(* Logix 5000 project; controller ACMI_PLC vendor 1 type 14 code 101 rev 19.11; software revision 19.01; part 2 of 18 *)

        [362].TIME.DAY := 6, [362].TIME.HOUR := 12, [362].TIME.MINUTE := 4, [362].TIME.SECOND := 14, [362].TIME.MICROSECOND := 99935, [362].EVENT := '2016/08/06   12:04:14   USER : PPS RESET FAULT BUTTON PRESSED', [363].TIME.YEAR := 2016, [363].TIME.MONTH := 8, [363].TIME.DAY := 6, [363].TIME.HOUR := 14, [363].TIME.MINUTE := 57, [363].TIME.SECOND := 32, [363].TIME.MICROSECOND := 599468, [363].EVENT := '2016/08/06   14:57:32   FAULT : QOW1 : Charge Outside Window Detected', [364].TIME.YEAR := 2016, [364].TIME.MONTH := 8, [364].TIME.DAY := 6, [364].TIME.HOUR := 14, [364].TIME.MINUTE := 57, [364].TIME.SECOND := 32, [364].TIME.MICROSECOND := 799580, [364].EVENT := '2016/08/06   14:57:32   USER : PPS RESET FAULT BUTTON PRESSED', [365].TIME.YEAR := 2016, [365].TIME.MONTH := 8, [365].TIME.DAY := 6, [365].TIME.HOUR := 14, [365].TIME.MINUTE := 57, [365].TIME.SECOND := 41, [365].TIME.MICROSECOND := 799582, [365].EVENT := '2016/08/06   14:57:41   USER : PPS RESET FAULT BUTTON PRESSED', [366].TIME.YEAR := 2016, [366].TIME.MONTH := 8, [366].TIME.DAY := 6, [366].TIME.HOUR := 14, [366].TIME.MINUTE := 57, [366].TIME.SECOND := 45, [366].TIME.MICROSECOND := 499509, [366].EVENT := '2016/08/06   14:57:45   USER : PPS RESET FAULT BUTTON PRESSED', [367].TIME.YEAR := 2016, [367].TIME.MONTH := 8, [367].TIME.DAY := 6, [367].TIME.HOUR := 18, [367].TIME.MINUTE := 23, [367].TIME.SECOND := 45, [367].TIME.MICROSECOND := 899510, [367].EVENT := '2016/08/06   18:23:45   USER : PPS RESET FAULT BUTTON PRESSED', [368].TIME.YEAR := 2016, [368].TIME.MONTH := 8, [368].TIME.DAY := 6, [368].TIME.HOUR := 18, [368].TIME.MINUTE := 28, [368].TIME.SECOND := 40, [368].TIME.MICROSECOND := 699977, [368].EVENT := '2016/08/06   18:28:40   FAULT : QOW1 : Charge Outside Window Detected', [369].TIME.YEAR := 2016, [369].TIME.MONTH := 8, [369].TIME.DAY := 6, [369].TIME.HOUR := 18, [369].TIME.MINUTE := 31, [369].TIME.SECOND := 49,
        [369].TIME.MICROSECOND := 299504, [369].EVENT := '2016/08/06   18:31:49   USER : PPS RESET FAULT BUTTON PRESSED', [370].TIME.YEAR := 2016, [370].TIME.MONTH := 8, [370].TIME.DAY := 7, [370].TIME.HOUR := 13, [370].TIME.MINUTE := 14, [370].TIME.SECOND := 49, [370].TIME.MICROSECOND := 699851, [370].EVENT := '2016/08/07   13:14:49   USER : PPS RESET FAULT BUTTON PRESSED', [371].TIME.YEAR := 2016, [371].TIME.MONTH := 8, [371].TIME.DAY := 7, [371].TIME.HOUR := 13, [371].TIME.MINUTE := 14, [371].TIME.SECOND := 53, [371].TIME.MICROSECOND := 399507, [371].EVENT := '2016/08/07   13:14:53   USER : PPS RESET FAULT BUTTON PRESSED', [372].TIME.YEAR := 2016, [372].TIME.MONTH := 8, [372].TIME.DAY := 7, [372].TIME.HOUR := 14, [372].TIME.MINUTE := 4, [372].TIME.SECOND := 34, [372].TIME.MICROSECOND := 499506, [372].EVENT := '2016/08/07   14:04:34   USER : PPS RESET FAULT BUTTON PRESSED', [373].TIME.YEAR := 2016, [373].TIME.MONTH := 8, [373].TIME.DAY := 7, [373].TIME.HOUR := 14, [373].TIME.MINUTE := 10, [373].TIME.SECOND := 33, [373].TIME.MICROSECOND := 599503, [373].EVENT := '2016/08/07   14:10:33   USER : PPS RESET FAULT BUTTON PRESSED', [374].TIME.YEAR := 2016, [374].TIME.MONTH := 8, [374].TIME.DAY := 7, [374].TIME.HOUR := 15, [374].TIME.MINUTE := 43, [374].TIME.SECOND := 5, [374].TIME.MICROSECOND := 599722, [374].EVENT := '2016/08/07   15:43:05   USER : PPS RESET FAULT BUTTON PRESSED', [375].TIME.YEAR := 2016, [375].TIME.MONTH := 8, [375].TIME.DAY := 7, [375].TIME.HOUR := 16, [375].TIME.MINUTE := 8, [375].TIME.SECOND := 27, [375].TIME.MICROSECOND := 699933, [375].EVENT := '2016/08/07   16:08:27   USER : PPS RESET FAULT BUTTON PRESSED', [376].TIME.YEAR := 2016, [376].TIME.MONTH := 8, [376].TIME.DAY := 7, [376].TIME.HOUR := 16, [376].TIME.MINUTE := 12, [376].TIME.SECOND := 25, [376].TIME.MICROSECOND := 299512, [376].EVENT := '2016/08/07   16:12:25   USER : PPS RESET FAULT BUTTON PRESSED', [377].TIME.YEAR := 2016, [377].TIME.MONTH := 8,
        [377].TIME.DAY := 7, [377].TIME.HOUR := 16, [377].TIME.MINUTE := 15, [377].TIME.SECOND := 37, [377].TIME.MICROSECOND := 299739, [377].EVENT := '2016/08/07   16:15:37   USER : PPS RESET FAULT BUTTON PRESSED', [378].TIME.YEAR := 2016, [378].TIME.MONTH := 8, [378].TIME.DAY := 7, [378].TIME.HOUR := 16, [378].TIME.MINUTE := 28, [378].TIME.SECOND := 37, [378].TIME.MICROSECOND := 299464, [378].EVENT := '2016/08/07   16:28:37   FAULT : QOW1 : Charge Outside Window Detected', [379].TIME.YEAR := 2016, [379].TIME.MONTH := 8, [379].TIME.DAY := 7, [379].TIME.HOUR := 16, [379].TIME.MINUTE := 29, [379].TIME.SECOND := 15, [379].TIME.MICROSECOND := 699509, [379].EVENT := '2016/08/07   16:29:15   USER : PPS RESET FAULT BUTTON PRESSED', [380].TIME.YEAR := 2016, [380].TIME.MONTH := 8, [380].TIME.DAY := 7, [380].TIME.HOUR := 16, [380].TIME.MINUTE := 29, [380].TIME.SECOND := 58, [380].TIME.MICROSECOND := 299502, [380].EVENT := '2016/08/07   16:29:58   USER : PPS RESET FAULT BUTTON PRESSED', [381].TIME.YEAR := 2016, [381].TIME.MONTH := 8, [381].TIME.DAY := 7, [381].TIME.HOUR := 17, [381].TIME.MINUTE := 7, [381].TIME.SECOND := 3, [381].TIME.MICROSECOND := 599449, [381].EVENT := '2016/08/07   17:07:03   FAULT : Storage Ring Accumulation HIGH', [382].TIME.YEAR := 2016, [382].TIME.MONTH := 8, [382].TIME.DAY := 7, [382].TIME.HOUR := 17, [382].TIME.MINUTE := 9, [382].TIME.SECOND := 13, [382].TIME.MICROSECOND := 499509, [382].EVENT := '2016/08/07   17:09:13   USER : PPS RESET FAULT BUTTON PRESSED', [383].TIME.YEAR := 2016, [383].TIME.MONTH := 8, [383].TIME.DAY := 7, [383].TIME.HOUR := 17, [383].TIME.MINUTE := 16, [383].TIME.SECOND := 23, [383].TIME.MICROSECOND := 799943, [383].EVENT := '2016/08/07   17:16:23   USER : PPS RESET FAULT BUTTON PRESSED', [384].TIME.YEAR := 2016, [384].TIME.MONTH := 8, [384].TIME.DAY := 7, [384].TIME.HOUR := 17, [384].TIME.MINUTE := 16, [384].TIME.SECOND := 25,
        [384].TIME.MICROSECOND := 699505, [384].EVENT := '2016/08/07   17:16:25   USER : PPS RESET FAULT BUTTON PRESSED', [385].TIME.YEAR := 2016, [385].TIME.MONTH := 8, [385].TIME.DAY := 7, [385].TIME.HOUR := 17, [385].TIME.MINUTE := 18, [385].TIME.SECOND := 4, [385].TIME.MICROSECOND := 899594, [385].EVENT := '2016/08/07   17:18:04   FAULT : Storage Ring Accumulation HIGH', [386].TIME.YEAR := 2016, [386].TIME.MONTH := 8, [386].TIME.DAY := 7, [386].TIME.HOUR := 17, [386].TIME.MINUTE := 18, [386].TIME.SECOND := 50, [386].TIME.MICROSECOND := 599506, [386].EVENT := '2016/08/07   17:18:50   USER : PPS RESET FAULT BUTTON PRESSED', [387].TIME.YEAR := 2016, [387].TIME.MONTH := 8, [387].TIME.DAY := 7, [387].TIME.HOUR := 17, [387].TIME.MINUTE := 20, [387].TIME.SECOND := 25, [387].TIME.MICROSECOND := 499450, [387].EVENT := '2016/08/07   17:20:25   FAULT : Storage Ring Accumulation HIGH', [388].TIME.YEAR := 2016, [388].TIME.MONTH := 8, [388].TIME.DAY := 7, [388].TIME.HOUR := 17, [388].TIME.MINUTE := 20, [388].TIME.SECOND := 25, [388].TIME.MICROSECOND := 699462, [388].EVENT := '2016/08/07   17:20:25   FAULT : QOW1 : Charge Outside Window Detected', [389].TIME.YEAR := 2016, [389].TIME.MONTH := 8, [389].TIME.DAY := 7, [389].TIME.HOUR := 17, [389].TIME.MINUTE := 21, [389].TIME.SECOND := 52, [389].TIME.MICROSECOND := 699506, [389].EVENT := '2016/08/07   17:21:52   USER : PPS RESET FAULT BUTTON PRESSED', [390].TIME.YEAR := 2016, [390].TIME.MONTH := 8, [390].TIME.DAY := 7, [390].TIME.HOUR := 17, [390].TIME.MINUTE := 30, [390].TIME.SECOND := 8, [390].TIME.MICROSECOND := 299449, [390].EVENT := '2016/08/07   17:30:08   FAULT : Storage Ring Accumulation HIGH', [391].TIME.YEAR := 2016, [391].TIME.MONTH := 8, [391].TIME.DAY := 7, [391].TIME.HOUR := 17, [391].TIME.MINUTE := 30, [391].TIME.SECOND := 53, [391].TIME.MICROSECOND := 299556, [391].EVENT := '2016/08/07   17:30:53   USER : PPS RESET FAULT BUTTON PRESSED', [392].TIME.YEAR := 2016, [392].TIME.MONTH := 8,
        [392].TIME.DAY := 7, [392].TIME.HOUR := 17, [392].TIME.MINUTE := 39, [392].TIME.SECOND := 26, [392].TIME.MICROSECOND := 699451, [392].EVENT := '2016/08/07   17:39:26   FAULT : Storage Ring Accumulation HIGH', [393].TIME.YEAR := 2016, [393].TIME.MONTH := 8, [393].TIME.DAY := 7, [393].TIME.HOUR := 17, [393].TIME.MINUTE := 40, [393].TIME.SECOND := 48, [393].TIME.MICROSECOND := 599508, [393].EVENT := '2016/08/07   17:40:48   USER : PPS RESET FAULT BUTTON PRESSED', [394].TIME.YEAR := 2016, [394].TIME.MONTH := 8, [394].TIME.DAY := 7, [394].TIME.HOUR := 17, [394].TIME.MINUTE := 40, [394].TIME.SECOND := 49, [394].TIME.MICROSECOND := 99507, [394].EVENT := '2016/08/07   17:40:49   USER : PPS RESET FAULT BUTTON PRESSED', [395].TIME.YEAR := 2016, [395].TIME.MONTH := 8, [395].TIME.DAY := 7, [395].TIME.HOUR := 17, [395].TIME.MINUTE := 52, [395].TIME.MICROSECOND := 599599, [395].EVENT := '2016/08/07   17:52:00   FAULT : Storage Ring Accumulation HIGH', [396].TIME.YEAR := 2016, [396].TIME.MONTH := 8, [396].TIME.DAY := 7, [396].TIME.HOUR := 17, [396].TIME.MINUTE := 53, [396].TIME.SECOND := 10, [396].TIME.MICROSECOND := 99562, [396].EVENT := '2016/08/07   17:53:10   USER : PPS RESET FAULT BUTTON PRESSED', [397].TIME.YEAR := 2016, [397].TIME.MONTH := 8, [397].TIME.DAY := 7, [397].TIME.HOUR := 18, [397].TIME.MICROSECOND := 999511, [397].EVENT := '2016/08/07   18:00:00   USER : PPS RESET FAULT BUTTON PRESSED', [398].TIME.YEAR := 2016, [398].TIME.MONTH := 8, [398].TIME.DAY := 7, [398].TIME.HOUR := 18, [398].TIME.SECOND := 51, [398].TIME.MICROSECOND := 499521, [398].EVENT := '2016/08/07   18:00:51   USER : PPS RESET FAULT BUTTON PRESSED', [399].TIME.YEAR := 2016, [399].TIME.MONTH := 8, [399].TIME.DAY := 7, [399].TIME.HOUR := 18, [399].TIME.MINUTE := 8, [399].TIME.SECOND := 30, [399].TIME.MICROSECOND := 299507, [399].EVENT := '2016/08/07   18:08:30   USER : PPS RESET FAULT BUTTON PRESSED', [400].TIME.YEAR := 2016, [400].TIME.MONTH := 8,
        [400].TIME.DAY := 8, [400].TIME.MINUTE := 42, [400].TIME.SECOND := 51, [400].TIME.MICROSECOND := 899938, [400].EVENT := '2016/08/08   00:42:51   USER : PPS RESET FAULT BUTTON PRESSED', [401].TIME.YEAR := 2016, [401].TIME.MONTH := 8, [401].TIME.DAY := 8, [401].TIME.HOUR := 1, [401].TIME.MINUTE := 23, [401].TIME.SECOND := 6, [401].TIME.MICROSECOND := 299510, [401].EVENT := '2016/08/08   01:23:06   USER : PPS RESET FAULT BUTTON PRESSED', [402].TIME.YEAR := 2016, [402].TIME.MONTH := 8, [402].TIME.DAY := 8, [402].TIME.HOUR := 4, [402].TIME.MINUTE := 37, [402].TIME.SECOND := 22, [402].TIME.MICROSECOND := 699521, [402].EVENT := '2016/08/08   04:37:22   USER : PPS RESET FAULT BUTTON PRESSED', [403].TIME.YEAR := 2016, [403].TIME.MONTH := 8, [403].TIME.DAY := 8, [403].TIME.HOUR := 8, [403].TIME.MINUTE := 26, [403].TIME.SECOND := 45, [403].TIME.MICROSECOND := 170, [403].EVENT := '2016/08/08   08:26:45   USER : PPS RESET FAULT BUTTON PRESSED', [404].TIME.YEAR := 2016, [404].TIME.MONTH := 8, [404].TIME.DAY := 8, [404].TIME.HOUR := 14, [404].TIME.MINUTE := 8, [404].TIME.SECOND := 27, [404].TIME.MICROSECOND := 399526, [404].EVENT := '2016/08/08   14:08:27   USER : PPS RESET FAULT BUTTON PRESSED', [405].TIME.YEAR := 2016, [405].TIME.MONTH := 8, [405].TIME.DAY := 8, [405].TIME.HOUR := 16, [405].TIME.MINUTE := 58, [405].TIME.SECOND := 17, [405].TIME.MICROSECOND := 299507, [405].EVENT := '2016/08/08   16:58:17   USER : PPS RESET FAULT BUTTON PRESSED', [406].TIME.YEAR := 2016, [406].TIME.MONTH := 8, [406].TIME.DAY := 8, [406].TIME.HOUR := 20, [406].TIME.MINUTE := 53, [406].TIME.SECOND := 34, [406].TIME.MICROSECOND := 99465, [406].EVENT := '2016/08/08   20:53:34   FAULT : QOW1 : Charge Outside Window Detected', [407].TIME.YEAR := 2016, [407].TIME.MONTH := 8, [407].TIME.DAY := 8, [407].TIME.HOUR := 20, [407].TIME.MINUTE := 53, [407].TIME.SECOND := 50, [407].TIME.MICROSECOND := 299514,
        [407].EVENT := '2016/08/08   20:53:50   USER : PPS RESET FAULT BUTTON PRESSED', [408].TIME.YEAR := 2016, [408].TIME.MONTH := 8, [408].TIME.DAY := 8, [408].TIME.HOUR := 21, [408].TIME.SECOND := 58, [408].TIME.MICROSECOND := 799510, [408].EVENT := '2016/08/08   21:00:58   USER : PPS RESET FAULT BUTTON PRESSED', [409].TIME.YEAR := 2016, [409].TIME.MONTH := 8, [409].TIME.DAY := 9, [409].TIME.HOUR := 16, [409].TIME.MINUTE := 51, [409].TIME.SECOND := 48, [409].TIME.MICROSECOND := 699509, [409].EVENT := '2016/08/09   16:51:48   USER : PPS RESET FAULT BUTTON PRESSED', [410].TIME.YEAR := 2016, [410].TIME.MONTH := 8, [410].TIME.DAY := 9, [410].TIME.HOUR := 16, [410].TIME.MINUTE := 52, [410].TIME.SECOND := 16, [410].TIME.MICROSECOND := 999461, [410].EVENT := '2016/08/09   16:52:16   FAULT : QOW1 : Charge Outside Window Detected', [411].TIME.YEAR := 2016, [411].TIME.MONTH := 8, [411].TIME.DAY := 9, [411].TIME.HOUR := 16, [411].TIME.MINUTE := 52, [411].TIME.SECOND := 51, [411].TIME.MICROSECOND := 199503, [411].EVENT := '2016/08/09   16:52:51   USER : PPS RESET FAULT BUTTON PRESSED', [412].TIME.YEAR := 2016, [412].TIME.MONTH := 8, [412].TIME.DAY := 9, [412].TIME.HOUR := 18, [412].TIME.MINUTE := 25, [412].TIME.SECOND := 25, [412].TIME.MICROSECOND := 799513, [412].EVENT := '2016/08/09   18:25:25   USER : PPS RESET FAULT BUTTON PRESSED', [413].TIME.YEAR := 2016, [413].TIME.MONTH := 8, [413].TIME.DAY := 9, [413].TIME.HOUR := 18, [413].TIME.MINUTE := 44, [413].TIME.SECOND := 50, [413].TIME.MICROSECOND := 600033, [413].EVENT := '2016/08/09   18:44:50   USER : PPS RESET FAULT BUTTON PRESSED', [414].TIME.YEAR := 2016, [414].TIME.MONTH := 8, [414].TIME.DAY := 9, [414].TIME.HOUR := 22, [414].TIME.MINUTE := 53, [414].TIME.SECOND := 46, [414].TIME.MICROSECOND := 999841, [414].EVENT := '2016/08/09   22:53:46   FAULT : QOW1 : Charge Outside Window Detected', [415].TIME.YEAR := 2016, [415].TIME.MONTH := 8, [415].TIME.DAY := 9, [415].TIME.HOUR := 22,
        [415].TIME.MINUTE := 54, [415].TIME.SECOND := 3, [415].TIME.MICROSECOND := 99504, [415].EVENT := '2016/08/09   22:54:03   USER : PPS RESET FAULT BUTTON PRESSED', [416].TIME.YEAR := 2016, [416].TIME.MONTH := 8, [416].TIME.DAY := 10, [416].TIME.HOUR := 4, [416].TIME.MINUTE := 15, [416].TIME.SECOND := 3, [416].TIME.MICROSECOND := 899896, [416].EVENT := '2016/08/10   04:15:03   FAULT : QOW1 : Charge Outside Window Detected', [417].TIME.YEAR := 2016, [417].TIME.MONTH := 8, [417].TIME.DAY := 10, [417].TIME.HOUR := 4, [417].TIME.MINUTE := 15, [417].TIME.SECOND := 18, [417].TIME.MICROSECOND := 799507, [417].EVENT := '2016/08/10   04:15:18   USER : PPS RESET FAULT BUTTON PRESSED', [418].TIME.YEAR := 2016, [418].TIME.MONTH := 8, [418].TIME.DAY := 10, [418].TIME.HOUR := 17, [418].TIME.MINUTE := 5, [418].TIME.SECOND := 50, [418].TIME.MICROSECOND := 799512, [418].EVENT := '2016/08/10   17:05:50   FAULT : QOW1 : Charge Outside Window Detected', [419].TIME.YEAR := 2016, [419].TIME.MONTH := 8, [419].TIME.DAY := 10, [419].TIME.HOUR := 17, [419].TIME.MINUTE := 5, [419].TIME.SECOND := 51, [419].TIME.MICROSECOND := 99507, [419].EVENT := '2016/08/10   17:05:51   USER : PPS RESET FAULT BUTTON PRESSED', [420].TIME.YEAR := 2016, [420].TIME.MONTH := 8, [420].TIME.DAY := 10, [420].TIME.HOUR := 17, [420].TIME.MINUTE := 6, [420].TIME.SECOND := 1, [420].TIME.MICROSECOND := 100028, [420].EVENT := '2016/08/10   17:06:01   USER : PPS RESET FAULT BUTTON PRESSED', [421].TIME.YEAR := 2016, [421].TIME.MONTH := 8, [421].TIME.DAY := 10, [421].TIME.HOUR := 17, [421].TIME.MINUTE := 8, [421].TIME.SECOND := 33, [421].TIME.MICROSECOND := 599516, [421].EVENT := '2016/08/10   17:08:33   USER : PPS RESET FAULT BUTTON PRESSED', [422].TIME.YEAR := 2016, [422].TIME.MONTH := 8, [422].TIME.DAY := 10, [422].TIME.HOUR := 17, [422].TIME.MINUTE := 33, [422].TIME.SECOND := 25, [422].TIME.MICROSECOND := 299511, [422].EVENT := '2016/08/10   17:33:25   USER : PPS RESET FAULT BUTTON PRESSED',
        [423].TIME.YEAR := 2016, [423].TIME.MONTH := 8, [423].TIME.DAY := 10, [423].TIME.HOUR := 17, [423].TIME.MINUTE := 46, [423].TIME.SECOND := 7, [423].TIME.MICROSECOND := 799463, [423].EVENT := '2016/08/10   17:46:07   FAULT : QOW1 : Charge Outside Window Detected', [424].TIME.YEAR := 2016, [424].TIME.MONTH := 8, [424].TIME.DAY := 10, [424].TIME.HOUR := 17, [424].TIME.MINUTE := 47, [424].TIME.SECOND := 1, [424].TIME.MICROSECOND := 599530, [424].EVENT := '2016/08/10   17:47:01   USER : PPS RESET FAULT BUTTON PRESSED', [425].TIME.YEAR := 2016, [425].TIME.MONTH := 8, [425].TIME.DAY := 11, [425].TIME.HOUR := 1, [425].TIME.MINUTE := 16, [425].TIME.SECOND := 30, [425].TIME.MICROSECOND := 999451, [425].EVENT := '2016/08/11   01:16:30   FAULT : Storage Ring Accumulation HIGH', [426].TIME.YEAR := 2016, [426].TIME.MONTH := 8, [426].TIME.DAY := 11, [426].TIME.HOUR := 1, [426].TIME.MINUTE := 16, [426].TIME.SECOND := 55, [426].TIME.MICROSECOND := 99506, [426].EVENT := '2016/08/11   01:16:55   USER : PPS RESET FAULT BUTTON PRESSED', [427].TIME.YEAR := 2016, [427].TIME.MONTH := 8, [427].TIME.DAY := 11, [427].TIME.HOUR := 5, [427].TIME.MINUTE := 52, [427].TIME.SECOND := 19, [427].TIME.MICROSECOND := 499510, [427].EVENT := '2016/08/11   05:52:19   USER : PPS RESET FAULT BUTTON PRESSED', [428].TIME.YEAR := 2016, [428].TIME.MONTH := 8, [428].TIME.DAY := 11, [428].TIME.HOUR := 6, [428].TIME.MINUTE := 51, [428].TIME.SECOND := 51, [428].TIME.MICROSECOND := 499508, [428].EVENT := '2016/08/11   06:51:51   USER : PPS RESET FAULT BUTTON PRESSED', [429].TIME.YEAR := 2016, [429].TIME.MONTH := 8, [429].TIME.DAY := 11, [429].TIME.HOUR := 13, [429].TIME.MINUTE := 21, [429].TIME.SECOND := 20, [429].TIME.MICROSECOND := 699504, [429].EVENT := '2016/08/11   13:21:20   USER : PPS RESET FAULT BUTTON PRESSED', [430].TIME.YEAR := 2016, [430].TIME.MONTH := 8, [430].TIME.DAY := 11, [430].TIME.HOUR := 14,
        [430].TIME.MINUTE := 4, [430].TIME.SECOND := 47, [430].TIME.MICROSECOND := 599502, [430].EVENT := '2016/08/11   14:04:47   USER : PPS RESET FAULT BUTTON PRESSED', [431].TIME.YEAR := 2016, [431].TIME.MONTH := 8, [431].TIME.DAY := 11, [431].TIME.HOUR := 15, [431].TIME.MINUTE := 12, [431].TIME.SECOND := 47, [431].TIME.MICROSECOND := 999508, [431].EVENT := '2016/08/11   15:12:47   USER : PPS RESET FAULT BUTTON PRESSED', [432].TIME.YEAR := 2016, [432].TIME.MONTH := 8, [432].TIME.DAY := 11, [432].TIME.HOUR := 19, [432].TIME.MINUTE := 47, [432].TIME.SECOND := 25, [432].TIME.MICROSECOND := 999651, [432].EVENT := '2016/08/11   19:47:25   USER : PPS RESET FAULT BUTTON PRESSED', [433].TIME.YEAR := 2016, [433].TIME.MONTH := 8, [433].TIME.DAY := 12, [433].TIME.HOUR := 2, [433].TIME.MINUTE := 31, [433].TIME.SECOND := 8, [433].TIME.MICROSECOND := 399504, [433].EVENT := '2016/08/12   02:31:08   USER : PPS RESET FAULT BUTTON PRESSED', [434].TIME.YEAR := 2016, [434].TIME.MONTH := 8, [434].TIME.DAY := 12, [434].TIME.HOUR := 16, [434].TIME.MINUTE := 21, [434].TIME.SECOND := 30, [434].TIME.MICROSECOND := 499936, [434].EVENT := '2016/08/12   16:21:30   USER : PPS RESET FAULT BUTTON PRESSED', [435].TIME.YEAR := 2016, [435].TIME.MONTH := 8, [435].TIME.DAY := 12, [435].TIME.HOUR := 16, [435].TIME.MINUTE := 21, [435].TIME.SECOND := 54, [435].TIME.MICROSECOND := 899511, [435].EVENT := '2016/08/12   16:21:54   USER : PPS RESET FAULT BUTTON PRESSED', [436].TIME.YEAR := 2016, [436].TIME.MONTH := 8, [436].TIME.DAY := 12, [436].TIME.HOUR := 16, [436].TIME.MINUTE := 24, [436].TIME.MICROSECOND := 99513, [436].EVENT := '2016/08/12   16:24:00   USER : PPS RESET FAULT BUTTON PRESSED', [437].TIME.YEAR := 2016, [437].TIME.MONTH := 8, [437].TIME.DAY := 12, [437].TIME.HOUR := 16, [437].TIME.MINUTE := 32, [437].TIME.SECOND := 10, [437].TIME.MICROSECOND := 99511, [437].EVENT := '2016/08/12   16:32:10   USER : PPS RESET FAULT BUTTON PRESSED', [438].TIME.YEAR := 2016,
        [438].TIME.MONTH := 8, [438].TIME.DAY := 12, [438].TIME.HOUR := 16, [438].TIME.MINUTE := 52, [438].TIME.SECOND := 35, [438].TIME.MICROSECOND := 999515, [438].EVENT := '2016/08/12   16:52:35   FAULT : QOW1 : Charge Outside Window Detected', [439].TIME.YEAR := 2016, [439].TIME.MONTH := 8, [439].TIME.DAY := 12, [439].TIME.HOUR := 16, [439].TIME.MINUTE := 57, [439].TIME.SECOND := 19, [439].TIME.MICROSECOND := 99507, [439].EVENT := '2016/08/12   16:57:19   USER : PPS RESET FAULT BUTTON PRESSED', [440].TIME.YEAR := 2016, [440].TIME.MONTH := 8, [440].TIME.DAY := 13, [440].TIME.HOUR := 10, [440].TIME.MINUTE := 42, [440].TIME.SECOND := 33, [440].TIME.MICROSECOND := 199466, [440].EVENT := '2016/08/13   10:42:33   FAULT : QOW1 : Charge Outside Window Detected', [441].TIME.YEAR := 2016, [441].TIME.MONTH := 8, [441].TIME.DAY := 13, [441].TIME.HOUR := 10, [441].TIME.MINUTE := 43, [441].TIME.SECOND := 44, [441].TIME.MICROSECOND := 299504, [441].EVENT := '2016/08/13   10:43:44   USER : PPS RESET FAULT BUTTON PRESSED', [442].TIME.YEAR := 2016, [442].TIME.MONTH := 8, [442].TIME.DAY := 13, [442].TIME.HOUR := 10, [442].TIME.MINUTE := 43, [442].TIME.SECOND := 46, [442].TIME.MICROSECOND := 499651, [442].EVENT := '2016/08/13   10:43:46   USER : PPS RESET FAULT BUTTON PRESSED', [443].TIME.YEAR := 2016, [443].TIME.MONTH := 8, [443].TIME.DAY := 13, [443].TIME.HOUR := 18, [443].TIME.MINUTE := 25, [443].TIME.SECOND := 45, [443].TIME.MICROSECOND := 200030, [443].EVENT := '2016/08/13   18:25:45   USER : PPS RESET FAULT BUTTON PRESSED', [444].TIME.YEAR := 2016, [444].TIME.MONTH := 8, [444].TIME.DAY := 13, [444].TIME.HOUR := 19, [444].TIME.MINUTE := 6, [444].TIME.SECOND := 5, [444].TIME.MICROSECOND := 499509, [444].EVENT := '2016/08/13   19:06:05   USER : PPS RESET FAULT BUTTON PRESSED', [445].TIME.YEAR := 2016, [445].TIME.MONTH := 8, [445].TIME.DAY := 13, [445].TIME.HOUR := 19, [445].TIME.MINUTE := 7,
        [445].TIME.SECOND := 19, [445].TIME.MICROSECOND := 899509, [445].EVENT := '2016/08/13   19:07:19   USER : PPS RESET FAULT BUTTON PRESSED', [446].TIME.YEAR := 2016, [446].TIME.MONTH := 8, [446].TIME.DAY := 13, [446].TIME.HOUR := 21, [446].TIME.MINUTE := 17, [446].TIME.SECOND := 33, [446].TIME.MICROSECOND := 699513, [446].EVENT := '2016/08/13   21:17:33   USER : PPS RESET FAULT BUTTON PRESSED', [447].TIME.YEAR := 2016, [447].TIME.MONTH := 8, [447].TIME.DAY := 14, [447].TIME.HOUR := 3, [447].TIME.MINUTE := 19, [447].TIME.SECOND := 29, [447].TIME.MICROSECOND := 199465, [447].EVENT := '2016/08/14   03:19:29   FAULT : QOW1 : Charge Outside Window Detected', [448].TIME.YEAR := 2016, [448].TIME.MONTH := 8, [448].TIME.DAY := 14, [448].TIME.HOUR := 3, [448].TIME.MINUTE := 30, [448].TIME.SECOND := 16, [448].TIME.MICROSECOND := 699503, [448].EVENT := '2016/08/14   03:30:16   USER : PPS RESET FAULT BUTTON PRESSED', [449].TIME.YEAR := 2016, [449].TIME.MONTH := 8, [449].TIME.DAY := 14, [449].TIME.HOUR := 3, [449].TIME.MINUTE := 38, [449].TIME.SECOND := 57, [449].TIME.MICROSECOND := 999680, [449].EVENT := '2016/08/14   03:38:57   USER : PPS RESET FAULT BUTTON PRESSED', [450].TIME.YEAR := 2016, [450].TIME.MONTH := 8, [450].TIME.DAY := 14, [450].TIME.HOUR := 3, [450].TIME.MINUTE := 39, [450].TIME.SECOND := 19, [450].TIME.MICROSECOND := 999887, [450].EVENT := '2016/08/14   03:39:19   FAULT : QOW1 : Charge Outside Window Detected', [451].TIME.YEAR := 2016, [451].TIME.MONTH := 8, [451].TIME.DAY := 14, [451].TIME.HOUR := 3, [451].TIME.MINUTE := 58, [451].TIME.SECOND := 14, [451].TIME.MICROSECOND := 499507, [451].EVENT := '2016/08/14   03:58:14   USER : PPS RESET FAULT BUTTON PRESSED', [452].TIME.YEAR := 2016, [452].TIME.MONTH := 8, [452].TIME.DAY := 14, [452].TIME.HOUR := 4, [452].TIME.MINUTE := 1, [452].TIME.SECOND := 42, [452].TIME.MICROSECOND := 999504, [452].EVENT := '2016/08/14   04:01:42   USER : PPS RESET FAULT BUTTON PRESSED', [453].TIME.YEAR := 2016,
        [453].TIME.MONTH := 8, [453].TIME.DAY := 14, [453].TIME.HOUR := 9, [453].TIME.MINUTE := 12, [453].TIME.SECOND := 1, [453].TIME.MICROSECOND := 399505, [453].EVENT := '2016/08/14   09:12:01   USER : PPS RESET FAULT BUTTON PRESSED', [454].TIME.YEAR := 2016, [454].TIME.MONTH := 8, [454].TIME.DAY := 14, [454].TIME.HOUR := 9, [454].TIME.MINUTE := 12, [454].TIME.SECOND := 5, [454].TIME.MICROSECOND := 799506, [454].EVENT := '2016/08/14   09:12:05   USER : PPS RESET FAULT BUTTON PRESSED', [455].TIME.YEAR := 2016, [455].TIME.MONTH := 8, [455].TIME.DAY := 14, [455].TIME.HOUR := 19, [455].TIME.MINUTE := 56, [455].TIME.SECOND := 57, [455].TIME.MICROSECOND := 899462, [455].EVENT := '2016/08/14   19:56:57   FAULT : QOW1 : Charge Outside Window Detected', [456].TIME.YEAR := 2016, [456].TIME.MONTH := 8, [456].TIME.DAY := 14, [456].TIME.HOUR := 19, [456].TIME.MINUTE := 58, [456].TIME.SECOND := 49, [456].TIME.MICROSECOND := 999510, [456].EVENT := '2016/08/14   19:58:49   USER : PPS RESET FAULT BUTTON PRESSED', [457].TIME.YEAR := 2016, [457].TIME.MONTH := 8, [457].TIME.DAY := 14, [457].TIME.HOUR := 19, [457].TIME.MINUTE := 58, [457].TIME.SECOND := 55, [457].TIME.MICROSECOND := 999511, [457].EVENT := '2016/08/14   19:58:55   USER : PPS RESET FAULT BUTTON PRESSED', [458].TIME.YEAR := 2016, [458].TIME.MONTH := 8, [458].TIME.DAY := 15, [458].TIME.HOUR := 4, [458].TIME.MINUTE := 21, [458].TIME.SECOND := 30, [458].TIME.MICROSECOND := 299561, [458].EVENT := '2016/08/15   04:21:30   USER : PPS RESET FAULT BUTTON PRESSED', [459].TIME.YEAR := 2016, [459].TIME.MONTH := 8, [459].TIME.DAY := 16, [459].TIME.HOUR := 14, [459].TIME.MINUTE := 25, [459].TIME.SECOND := 39, [459].TIME.MICROSECOND := 699467, [459].EVENT := '2016/08/16   14:25:39   FAULT : QOW1 : Charge Outside Window Detected', [460].TIME.YEAR := 2016, [460].TIME.MONTH := 8, [460].TIME.DAY := 16, [460].TIME.HOUR := 14, [460].TIME.MINUTE := 25,
        [460].TIME.SECOND := 51, [460].TIME.MICROSECOND := 899506, [460].EVENT := '2016/08/16   14:25:51   USER : PPS RESET FAULT BUTTON PRESSED', [461].TIME.YEAR := 2016, [461].TIME.MONTH := 8, [461].TIME.DAY := 17, [461].TIME.HOUR := 9, [461].TIME.MINUTE := 19, [461].TIME.SECOND := 27, [461].TIME.MICROSECOND := 800026, [461].EVENT := '2016/08/17   09:19:27   USER : PPS RESET FAULT BUTTON PRESSED', [462].TIME.YEAR := 2016, [462].TIME.MONTH := 8, [462].TIME.DAY := 17, [462].TIME.HOUR := 9, [462].TIME.MINUTE := 29, [462].TIME.SECOND := 22, [462].TIME.MICROSECOND := 699555, [462].EVENT := '2016/08/17   09:29:22   USER : PPS RESET FAULT BUTTON PRESSED', [463].TIME.YEAR := 2016, [463].TIME.MONTH := 8, [463].TIME.DAY := 17, [463].TIME.HOUR := 9, [463].TIME.MINUTE := 30, [463].TIME.SECOND := 56, [463].TIME.MICROSECOND := 499725, [463].EVENT := '2016/08/17   09:30:56   USER : PPS RESET FAULT BUTTON PRESSED', [464].TIME.YEAR := 2016, [464].TIME.MONTH := 8, [464].TIME.DAY := 17, [464].TIME.HOUR := 9, [464].TIME.MINUTE := 45, [464].TIME.SECOND := 1, [464].TIME.MICROSECOND := 599506, [464].EVENT := '2016/08/17   09:45:01   USER : PPS RESET FAULT BUTTON PRESSED', [465].TIME.YEAR := 2016, [465].TIME.MONTH := 8, [465].TIME.DAY := 17, [465].TIME.HOUR := 10, [465].TIME.MINUTE := 8, [465].TIME.SECOND := 31, [465].TIME.MICROSECOND := 299511, [465].EVENT := '2016/08/17   10:08:31   USER : PPS RESET FAULT BUTTON PRESSED', [466].TIME.YEAR := 2016, [466].TIME.MONTH := 8, [466].TIME.DAY := 17, [466].TIME.HOUR := 10, [466].TIME.MINUTE := 12, [466].TIME.SECOND := 27, [466].TIME.MICROSECOND := 299510, [466].EVENT := '2016/08/17   10:12:27   USER : PPS RESET FAULT BUTTON PRESSED', [467].TIME.YEAR := 2016, [467].TIME.MONTH := 8, [467].TIME.DAY := 17, [467].TIME.HOUR := 10, [467].TIME.MINUTE := 12, [467].TIME.SECOND := 30, [467].TIME.MICROSECOND := 399508, [467].EVENT := '2016/08/17   10:12:30   USER : PPS RESET FAULT BUTTON PRESSED', [468].TIME.YEAR := 2016,
        [468].TIME.MONTH := 8, [468].TIME.DAY := 17, [468].TIME.HOUR := 10, [468].TIME.MINUTE := 12, [468].TIME.SECOND := 36, [468].TIME.MICROSECOND := 900030, [468].EVENT := '2016/08/17   10:12:36   USER : PPS RESET FAULT BUTTON PRESSED', [469].TIME.YEAR := 2016, [469].TIME.MONTH := 8, [469].TIME.DAY := 17, [469].TIME.HOUR := 10, [469].TIME.MINUTE := 17, [469].TIME.SECOND := 56, [469].TIME.MICROSECOND := 599509, [469].EVENT := '2016/08/17   10:17:56   USER : PPS RESET FAULT BUTTON PRESSED', [470].TIME.YEAR := 2016, [470].TIME.MONTH := 8, [470].TIME.DAY := 17, [470].TIME.HOUR := 11, [470].TIME.MINUTE := 20, [470].TIME.SECOND := 16, [470].TIME.MICROSECOND := 599503, [470].EVENT := '2016/08/17   11:20:16   USER : PPS RESET FAULT BUTTON PRESSED', [471].TIME.YEAR := 2016, [471].TIME.MONTH := 8, [471].TIME.DAY := 17, [471].TIME.HOUR := 11, [471].TIME.MINUTE := 20, [471].TIME.SECOND := 24, [471].TIME.MICROSECOND := 199526, [471].EVENT := '2016/08/17   11:20:24   USER : PPS RESET FAULT BUTTON PRESSED', [472].TIME.YEAR := 2016, [472].TIME.MONTH := 8, [472].TIME.DAY := 17, [472].TIME.HOUR := 11, [472].TIME.MINUTE := 22, [472].TIME.SECOND := 56, [472].TIME.MICROSECOND := 499504, [472].EVENT := '2016/08/17   11:22:56   USER : PPS RESET FAULT BUTTON PRESSED', [473].TIME.YEAR := 2016, [473].TIME.MONTH := 8, [473].TIME.DAY := 17, [473].TIME.HOUR := 11, [473].TIME.MINUTE := 24, [473].TIME.SECOND := 41, [473].TIME.MICROSECOND := 499557, [473].EVENT := '2016/08/17   11:24:41   USER : PPS RESET FAULT BUTTON PRESSED', [474].TIME.YEAR := 2016, [474].TIME.MONTH := 8, [474].TIME.DAY := 17, [474].TIME.HOUR := 13, [474].TIME.MINUTE := 2, [474].TIME.SECOND := 51, [474].TIME.MICROSECOND := 199488, [474].EVENT := '2016/08/17   13:02:51   FAULT : QOW1 : Charge Outside Window Detected', [475].TIME.YEAR := 2016, [475].TIME.MONTH := 8, [475].TIME.DAY := 17, [475].TIME.HOUR := 13, [475].TIME.MINUTE := 9,
        [475].TIME.SECOND := 21, [475].TIME.MICROSECOND := 500025, [475].EVENT := '2016/08/17   13:09:21   USER : PPS RESET FAULT BUTTON PRESSED', [476].TIME.YEAR := 2016, [476].TIME.MONTH := 8, [476].TIME.DAY := 17, [476].TIME.HOUR := 16, [476].TIME.MINUTE := 31, [476].TIME.SECOND := 24, [476].TIME.MICROSECOND := 999509, [476].EVENT := '2016/08/17   16:31:24   USER : PPS RESET FAULT BUTTON PRESSED', [477].TIME.YEAR := 2016, [477].TIME.MONTH := 8, [477].TIME.DAY := 17, [477].TIME.HOUR := 16, [477].TIME.MINUTE := 40, [477].TIME.SECOND := 51, [477].TIME.MICROSECOND := 299937, [477].EVENT := '2016/08/17   16:40:51   USER : PPS RESET FAULT BUTTON PRESSED', [478].TIME.YEAR := 2016, [478].TIME.MONTH := 8, [478].TIME.DAY := 17, [478].TIME.HOUR := 16, [478].TIME.MINUTE := 45, [478].TIME.SECOND := 7, [478].TIME.MICROSECOND := 199517, [478].EVENT := '2016/08/17   16:45:07   USER : PPS RESET FAULT BUTTON PRESSED', [479].TIME.YEAR := 2016, [479].TIME.MONTH := 8, [479].TIME.DAY := 17, [479].TIME.HOUR := 16, [479].TIME.MINUTE := 58, [479].TIME.SECOND := 20, [479].TIME.MICROSECOND := 899461, [479].EVENT := '2016/08/17   16:58:20   FAULT : QOW1 : Charge Outside Window Detected', [480].TIME.YEAR := 2016, [480].TIME.MONTH := 8, [480].TIME.DAY := 17, [480].TIME.HOUR := 17, [480].TIME.MINUTE := 2, [480].TIME.SECOND := 11, [480].TIME.MICROSECOND := 499503, [480].EVENT := '2016/08/17   17:02:11   USER : PPS RESET FAULT BUTTON PRESSED', [481].TIME.YEAR := 2016, [481].TIME.MONTH := 8, [481].TIME.DAY := 17, [481].TIME.HOUR := 17, [481].TIME.MINUTE := 2, [481].TIME.SECOND := 12, [481].TIME.MICROSECOND := 399510, [481].EVENT := '2016/08/17   17:02:12   USER : PPS RESET FAULT BUTTON PRESSED', [482].TIME.YEAR := 2016, [482].TIME.MONTH := 8, [482].TIME.DAY := 17, [482].TIME.HOUR := 17, [482].TIME.MINUTE := 32, [482].TIME.SECOND := 54, [482].TIME.MICROSECOND := 299505, [482].EVENT := '2016/08/17   17:32:54   USER : PPS RESET FAULT BUTTON PRESSED', [483].TIME.YEAR := 2016,
        [483].TIME.MONTH := 8, [483].TIME.DAY := 17, [483].TIME.HOUR := 17, [483].TIME.MINUTE := 34, [483].TIME.SECOND := 9, [483].TIME.MICROSECOND := 699506, [483].EVENT := '2016/08/17   17:34:09   USER : PPS RESET FAULT BUTTON PRESSED', [484].TIME.YEAR := 2016, [484].TIME.MONTH := 8, [484].TIME.DAY := 17, [484].TIME.HOUR := 18, [484].TIME.MINUTE := 32, [484].TIME.SECOND := 24, [484].TIME.MICROSECOND := 99507, [484].EVENT := '2016/08/17   18:32:24   USER : PPS RESET FAULT BUTTON PRESSED', [485].TIME.YEAR := 2016, [485].TIME.MONTH := 8, [485].TIME.DAY := 17, [485].TIME.HOUR := 20, [485].TIME.MINUTE := 51, [485].TIME.SECOND := 28, [485].TIME.MICROSECOND := 899507, [485].EVENT := '2016/08/17   20:51:28   USER : PPS RESET FAULT BUTTON PRESSED', [486].TIME.YEAR := 2016, [486].TIME.MONTH := 8, [486].TIME.DAY := 18, [486].TIME.MINUTE := 22, [486].TIME.SECOND := 47, [486].TIME.MICROSECOND := 799507, [486].EVENT := '2016/08/18   00:22:47   USER : PPS RESET FAULT BUTTON PRESSED', [487].TIME.YEAR := 2016, [487].TIME.MONTH := 8, [487].TIME.DAY := 18, [487].TIME.HOUR := 5, [487].TIME.MINUTE := 45, [487].TIME.SECOND := 44, [487].TIME.MICROSECOND := 399510, [487].EVENT := '2016/08/18   05:45:44   USER : PPS RESET FAULT BUTTON PRESSED', [488].TIME.YEAR := 2016, [488].TIME.MONTH := 8, [488].TIME.DAY := 18, [488].TIME.HOUR := 5, [488].TIME.MINUTE := 53, [488].TIME.SECOND := 55, [488].TIME.MICROSECOND := 599934, [488].EVENT := '2016/08/18   05:53:55   USER : PPS RESET FAULT BUTTON PRESSED', [489].TIME.YEAR := 2016, [489].TIME.MONTH := 8, [489].TIME.DAY := 18, [489].TIME.HOUR := 6, [489].TIME.MINUTE := 14, [489].TIME.SECOND := 56, [489].TIME.MICROSECOND := 599506, [489].EVENT := '2016/08/18   06:14:56   USER : PPS RESET FAULT BUTTON PRESSED', [490].TIME.YEAR := 2016, [490].TIME.MONTH := 8, [490].TIME.DAY := 18, [490].TIME.HOUR := 6, [490].TIME.MINUTE := 14, [490].TIME.SECOND := 58,
        [490].TIME.MICROSECOND := 99512, [490].EVENT := '2016/08/18   06:14:58   USER : PPS RESET FAULT BUTTON PRESSED', [491].TIME.YEAR := 2016, [491].TIME.MONTH := 8, [491].TIME.DAY := 18, [491].TIME.HOUR := 6, [491].TIME.MINUTE := 15, [491].TIME.SECOND := 1, [491].TIME.MICROSECOND := 999506, [491].EVENT := '2016/08/18   06:15:01   USER : PPS RESET FAULT BUTTON PRESSED', [492].TIME.YEAR := 2016, [492].TIME.MONTH := 8, [492].TIME.DAY := 18, [492].TIME.HOUR := 6, [492].TIME.MINUTE := 39, [492].TIME.SECOND := 58, [492].TIME.MICROSECOND := 799939, [492].EVENT := '2016/08/18   06:39:58   USER : PPS RESET FAULT BUTTON PRESSED', [493].TIME.YEAR := 2016, [493].TIME.MONTH := 8, [493].TIME.DAY := 19, [493].TIME.HOUR := 2, [493].TIME.MINUTE := 29, [493].TIME.SECOND := 21, [493].TIME.MICROSECOND := 599508, [493].EVENT := '2016/08/19   02:29:21   USER : PPS RESET FAULT BUTTON PRESSED', [494].TIME.YEAR := 2016, [494].TIME.MONTH := 8, [494].TIME.DAY := 19, [494].TIME.HOUR := 8, [494].TIME.MINUTE := 25, [494].TIME.SECOND := 13, [494].TIME.MICROSECOND := 299504, [494].EVENT := '2016/08/19   08:25:13   USER : PPS RESET FAULT BUTTON PRESSED', [495].TIME.YEAR := 2016, [495].TIME.MONTH := 8, [495].TIME.DAY := 19, [495].TIME.HOUR := 8, [495].TIME.MINUTE := 25, [495].TIME.SECOND := 19, [495].TIME.MICROSECOND := 799509, [495].EVENT := '2016/08/19   08:25:19   USER : PPS RESET FAULT BUTTON PRESSED', [496].TIME.YEAR := 2016, [496].TIME.MONTH := 8, [496].TIME.DAY := 20, [496].TIME.HOUR := 11, [496].TIME.MINUTE := 43, [496].TIME.SECOND := 48, [496].TIME.MICROSECOND := 299512, [496].EVENT := '2016/08/20   11:43:48   USER : PPS RESET FAULT BUTTON PRESSED', [497].TIME.YEAR := 2016, [497].TIME.MONTH := 8, [497].TIME.DAY := 21, [497].TIME.HOUR := 14, [497].TIME.MINUTE := 35, [497].TIME.SECOND := 36, [497].TIME.MICROSECOND := 599525, [497].EVENT := '2016/08/21   14:35:36   USER : PPS RESET FAULT BUTTON PRESSED', [498].TIME.YEAR := 2016, [498].TIME.MONTH := 8,
        [498].TIME.DAY := 21, [498].TIME.HOUR := 14, [498].TIME.MINUTE := 36, [498].TIME.SECOND := 48, [498].TIME.MICROSECOND := 700027, [498].EVENT := '2016/08/21   14:36:48   USER : PPS RESET FAULT BUTTON PRESSED', [499].TIME.YEAR := 2016, [499].TIME.MONTH := 8, [499].TIME.DAY := 24, [499].TIME.HOUR := 7, [499].TIME.MINUTE := 15, [499].TIME.SECOND := 5, [499].TIME.MICROSECOND := 299509, [499].EVENT := '2016/08/24   07:15:05   USER : PPS RESET FAULT BUTTON PRESSED', [500].TIME.YEAR := 2016, [500].TIME.MONTH := 8, [500].TIME.DAY := 24, [500].TIME.HOUR := 9, [500].TIME.MINUTE := 26, [500].TIME.SECOND := 32, [500].TIME.MICROSECOND := 699510, [500].EVENT := '2016/08/24   09:26:32   USER : PPS RESET FAULT BUTTON PRESSED', [501].TIME.YEAR := 2016, [501].TIME.MONTH := 8, [501].TIME.DAY := 25, [501].TIME.HOUR := 10, [501].TIME.MINUTE := 44, [501].TIME.SECOND := 49, [501].TIME.MICROSECOND := 599509, [501].EVENT := '2016/08/25   10:44:49   USER : PPS RESET FAULT BUTTON PRESSED', [502].TIME.YEAR := 2016, [502].TIME.MONTH := 8, [502].TIME.DAY := 25, [502].TIME.HOUR := 10, [502].TIME.MINUTE := 54, [502].TIME.SECOND := 15, [502].TIME.MICROSECOND := 999556, [502].EVENT := '2016/08/25   10:54:15   USER : PPS RESET FAULT BUTTON PRESSED', [503].TIME.YEAR := 2016, [503].TIME.MONTH := 8, [503].TIME.DAY := 26, [503].TIME.HOUR := 6, [503].TIME.MINUTE := 55, [503].TIME.SECOND := 43, [503].TIME.MICROSECOND := 199455, [503].EVENT := '2016/08/26   06:55:43   FAULT : QOW1 : Charge Outside Window Detected', [504].TIME.YEAR := 2016, [504].TIME.MONTH := 8, [504].TIME.DAY := 26, [504].TIME.HOUR := 7, [504].TIME.MINUTE := 1, [504].TIME.SECOND := 12, [504].TIME.MICROSECOND := 899508, [504].EVENT := '2016/08/26   07:01:12   USER : PPS RESET FAULT BUTTON PRESSED', [505].TIME.YEAR := 2016, [505].TIME.MONTH := 8, [505].TIME.DAY := 26, [505].TIME.HOUR := 13, [505].TIME.MINUTE := 12, [505].TIME.SECOND := 40,
        [505].TIME.MICROSECOND := 800023, [505].EVENT := '2016/08/26   13:12:40   USER : PPS RESET FAULT BUTTON PRESSED', [506].TIME.YEAR := 2016, [506].TIME.MONTH := 8, [506].TIME.DAY := 26, [506].TIME.HOUR := 13, [506].TIME.MINUTE := 12, [506].TIME.SECOND := 46, [506].TIME.MICROSECOND := 499508, [506].EVENT := '2016/08/26   13:12:46   USER : PPS RESET FAULT BUTTON PRESSED', [507].TIME.YEAR := 2016, [507].TIME.MONTH := 8, [507].TIME.DAY := 26, [507].TIME.HOUR := 15, [507].TIME.MINUTE := 2, [507].TIME.SECOND := 26, [507].TIME.MICROSECOND := 99506, [507].EVENT := '2016/08/26   15:02:26   USER : PPS RESET FAULT BUTTON PRESSED', [508].TIME.YEAR := 2016, [508].TIME.MONTH := 8, [508].TIME.DAY := 26, [508].TIME.HOUR := 17, [508].TIME.MINUTE := 15, [508].TIME.SECOND := 6, [508].TIME.MICROSECOND := 299467, [508].EVENT := '2016/08/26   17:15:06   FAULT : QOW1 : Charge Outside Window Detected', [509].TIME.YEAR := 2016, [509].TIME.MONTH := 8, [509].TIME.DAY := 26, [509].TIME.HOUR := 17, [509].TIME.MINUTE := 17, [509].TIME.SECOND := 35, [509].TIME.MICROSECOND := 299516, [509].EVENT := '2016/08/26   17:17:35   USER : PPS RESET FAULT BUTTON PRESSED', [510].TIME.YEAR := 2016, [510].TIME.MONTH := 8, [510].TIME.DAY := 26, [510].TIME.HOUR := 19, [510].TIME.MINUTE := 32, [510].TIME.SECOND := 38, [510].TIME.MICROSECOND := 299512, [510].EVENT := '2016/08/26   19:32:38   USER : PPS RESET FAULT BUTTON PRESSED', [511].TIME.YEAR := 2016, [511].TIME.MONTH := 8, [511].TIME.DAY := 26, [511].TIME.HOUR := 20, [511].TIME.MINUTE := 22, [511].TIME.SECOND := 31, [511].TIME.MICROSECOND := 599539, [511].EVENT := '2016/08/26   20:22:31   USER : PPS RESET FAULT BUTTON PRESSED', [512].TIME.YEAR := 2016, [512].TIME.MONTH := 8, [512].TIME.DAY := 26, [512].TIME.HOUR := 20, [512].TIME.MINUTE := 22, [512].TIME.SECOND := 36, [512].TIME.MICROSECOND := 499511, [512].EVENT := '2016/08/26   20:22:36   USER : PPS RESET FAULT BUTTON PRESSED', [513].TIME.YEAR := 2016, [513].TIME.MONTH := 8,
        [513].TIME.DAY := 26, [513].TIME.HOUR := 20, [513].TIME.MINUTE := 22, [513].TIME.SECOND := 41, [513].TIME.MICROSECOND := 199508, [513].EVENT := '2016/08/26   20:22:41   USER : PPS RESET FAULT BUTTON PRESSED', [514].TIME.YEAR := 2016, [514].TIME.MONTH := 8, [514].TIME.DAY := 27, [514].TIME.HOUR := 8, [514].TIME.MINUTE := 35, [514].TIME.SECOND := 33, [514].TIME.MICROSECOND := 599508, [514].EVENT := '2016/08/27   08:35:33   USER : PPS RESET FAULT BUTTON PRESSED', [515].TIME.YEAR := 2016, [515].TIME.MONTH := 8, [515].TIME.DAY := 27, [515].TIME.HOUR := 8, [515].TIME.MINUTE := 54, [515].TIME.SECOND := 32, [515].TIME.MICROSECOND := 799511, [515].EVENT := '2016/08/27   08:54:32   USER : PPS RESET FAULT BUTTON PRESSED', [516].TIME.YEAR := 2016, [516].TIME.MONTH := 8, [516].TIME.DAY := 27, [516].TIME.HOUR := 11, [516].TIME.MINUTE := 37, [516].TIME.SECOND := 4, [516].TIME.MICROSECOND := 899933, [516].EVENT := '2016/08/27   11:37:04   USER : PPS RESET FAULT BUTTON PRESSED', [517].TIME.YEAR := 2016, [517].TIME.MONTH := 8, [517].TIME.DAY := 27, [517].TIME.HOUR := 11, [517].TIME.MINUTE := 44, [517].TIME.SECOND := 12, [517].TIME.MICROSECOND := 599513, [517].EVENT := '2016/08/27   11:44:12   USER : PPS RESET FAULT BUTTON PRESSED', [518].TIME.YEAR := 2016, [518].TIME.MONTH := 8, [518].TIME.DAY := 27, [518].TIME.HOUR := 16, [518].TIME.MINUTE := 22, [518].TIME.SECOND := 19, [518].TIME.MICROSECOND := 799506, [518].EVENT := '2016/08/27   16:22:19   USER : PPS RESET FAULT BUTTON PRESSED', [519].TIME.YEAR := 2016, [519].TIME.MONTH := 8, [519].TIME.DAY := 27, [519].TIME.HOUR := 16, [519].TIME.MINUTE := 22, [519].TIME.SECOND := 20, [519].TIME.MICROSECOND := 99511, [519].EVENT := '2016/08/27   16:22:20   USER : PPS RESET FAULT BUTTON PRESSED', [520].TIME.YEAR := 2016, [520].TIME.MONTH := 8, [520].TIME.DAY := 27, [520].TIME.HOUR := 16, [520].TIME.MINUTE := 22, [520].TIME.SECOND := 20,
        [520].TIME.MICROSECOND := 299504, [520].EVENT := '2016/08/27   16:22:20   USER : PPS RESET FAULT BUTTON PRESSED', [521].TIME.YEAR := 2016, [521].TIME.MONTH := 8, [521].TIME.DAY := 27, [521].TIME.HOUR := 16, [521].TIME.MINUTE := 37, [521].TIME.SECOND := 9, [521].TIME.MICROSECOND := 799509, [521].EVENT := '2016/08/27   16:37:09   USER : PPS RESET FAULT BUTTON PRESSED', [522].TIME.YEAR := 2016, [522].TIME.MONTH := 8, [522].TIME.DAY := 27, [522].TIME.HOUR := 16, [522].TIME.MINUTE := 39, [522].TIME.SECOND := 25, [522].TIME.MICROSECOND := 699937, [522].EVENT := '2016/08/27   16:39:25   USER : PPS RESET FAULT BUTTON PRESSED', [523].TIME.YEAR := 2016, [523].TIME.MONTH := 8, [523].TIME.DAY := 27, [523].TIME.HOUR := 16, [523].TIME.MINUTE := 44, [523].TIME.SECOND := 27, [523].TIME.MICROSECOND := 199457, [523].EVENT := '2016/08/27   16:44:27   FAULT : QOW1 : Charge Outside Window Detected', [524].TIME.YEAR := 2016, [524].TIME.MONTH := 8, [524].TIME.DAY := 27, [524].TIME.HOUR := 16, [524].TIME.MINUTE := 45, [524].TIME.SECOND := 35, [524].TIME.MICROSECOND := 600017, [524].EVENT := '2016/08/27   16:45:35   USER : PPS RESET FAULT BUTTON PRESSED', [525].TIME.YEAR := 2016, [525].TIME.MONTH := 8, [525].TIME.DAY := 27, [525].TIME.HOUR := 16, [525].TIME.MINUTE := 45, [525].TIME.SECOND := 37, [525].TIME.MICROSECOND := 399510, [525].EVENT := '2016/08/27   16:45:37   USER : PPS RESET FAULT BUTTON PRESSED', [526].TIME.YEAR := 2016, [526].TIME.MONTH := 8, [526].TIME.DAY := 27, [526].TIME.HOUR := 16, [526].TIME.MINUTE := 55, [526].TIME.SECOND := 5, [526].TIME.MICROSECOND := 499520, [526].EVENT := '2016/08/27   16:55:05   USER : PPS RESET FAULT BUTTON PRESSED', [527].TIME.YEAR := 2016, [527].TIME.MONTH := 8, [527].TIME.DAY := 28, [527].TIME.HOUR := 1, [527].TIME.MINUTE := 19, [527].TIME.SECOND := 35, [527].TIME.MICROSECOND := 799466, [527].EVENT := '2016/08/28   01:19:35   FAULT : QOW1 : Charge Outside Window Detected', [528].TIME.YEAR := 2016, [528].TIME.MONTH := 8,
        [528].TIME.DAY := 28, [528].TIME.HOUR := 1, [528].TIME.MINUTE := 21, [528].TIME.SECOND := 56, [528].TIME.MICROSECOND := 399503, [528].EVENT := '2016/08/28   01:21:56   USER : PPS RESET FAULT BUTTON PRESSED', [529].TIME.YEAR := 2016, [529].TIME.MONTH := 8, [529].TIME.DAY := 28, [529].TIME.HOUR := 3, [529].TIME.MINUTE := 50, [529].TIME.SECOND := 19, [529].TIME.MICROSECOND := 599890, [529].EVENT := '2016/08/28   03:50:19   FAULT : QOW1 : Charge Outside Window Detected', [530].TIME.YEAR := 2016, [530].TIME.MONTH := 8, [530].TIME.DAY := 28, [530].TIME.HOUR := 4, [530].TIME.MINUTE := 2, [530].TIME.SECOND := 44, [530].TIME.MICROSECOND := 599507, [530].EVENT := '2016/08/28   04:02:44   USER : PPS RESET FAULT BUTTON PRESSED', [531].TIME.YEAR := 2016, [531].TIME.MONTH := 8, [531].TIME.DAY := 28, [531].TIME.HOUR := 6, [531].TIME.MINUTE := 35, [531].TIME.SECOND := 39, [531].TIME.MICROSECOND := 99664, [531].EVENT := '2016/08/28   06:35:39   USER : PPS RESET FAULT BUTTON PRESSED', [532].TIME.YEAR := 2016, [532].TIME.MONTH := 8, [532].TIME.DAY := 28, [532].TIME.HOUR := 6, [532].TIME.MINUTE := 39, [532].TIME.SECOND := 44, [532].TIME.MICROSECOND := 399505, [532].EVENT := '2016/08/28   06:39:44   USER : PPS RESET FAULT BUTTON PRESSED', [533].TIME.YEAR := 2016, [533].TIME.MONTH := 8, [533].TIME.DAY := 28, [533].TIME.HOUR := 12, [533].TIME.MINUTE := 23, [533].TIME.SECOND := 29, [533].TIME.MICROSECOND := 199512, [533].EVENT := '2016/08/28   12:23:29   USER : PPS RESET FAULT BUTTON PRESSED', [534].TIME.YEAR := 2016, [534].TIME.MONTH := 8, [534].TIME.DAY := 28, [534].TIME.HOUR := 13, [534].TIME.MINUTE := 57, [534].TIME.SECOND := 37, [534].TIME.MICROSECOND := 899651, [534].EVENT := '2016/08/28   13:57:37   USER : PPS RESET FAULT BUTTON PRESSED', [535].TIME.YEAR := 2016, [535].TIME.MONTH := 8, [535].TIME.DAY := 28, [535].TIME.HOUR := 19, [535].TIME.MINUTE := 17, [535].TIME.SECOND := 36,
        [535].TIME.MICROSECOND := 499513, [535].EVENT := '2016/08/28   19:17:36   USER : PPS RESET FAULT BUTTON PRESSED', [536].TIME.YEAR := 2016, [536].TIME.MONTH := 8, [536].TIME.DAY := 29, [536].TIME.MINUTE := 36, [536].TIME.SECOND := 49, [536].TIME.MICROSECOND := 99465, [536].EVENT := '2016/08/29   00:36:49   FAULT : QOW1 : Charge Outside Window Detected', [537].TIME.YEAR := 2016, [537].TIME.MONTH := 8, [537].TIME.DAY := 29, [537].TIME.MINUTE := 38, [537].TIME.SECOND := 5, [537].TIME.MICROSECOND := 999508, [537].EVENT := '2016/08/29   00:38:05   USER : PPS RESET FAULT BUTTON PRESSED', [538].TIME.YEAR := 2016, [538].TIME.MONTH := 8, [538].TIME.DAY := 29, [538].TIME.HOUR := 12, [538].TIME.MINUTE := 44, [538].TIME.SECOND := 43, [538].TIME.MICROSECOND := 199510, [538].EVENT := '2016/08/29   12:44:43   USER : PPS RESET FAULT BUTTON PRESSED', [539].TIME.YEAR := 2016, [539].TIME.MONTH := 8, [539].TIME.DAY := 29, [539].TIME.HOUR := 13, [539].TIME.MINUTE := 29, [539].TIME.SECOND := 13, [539].TIME.MICROSECOND := 499936, [539].EVENT := '2016/08/29   13:29:13   USER : PPS RESET FAULT BUTTON PRESSED', [540].TIME.YEAR := 2016, [540].TIME.MONTH := 8, [540].TIME.DAY := 29, [540].TIME.HOUR := 13, [540].TIME.MINUTE := 43, [540].TIME.SECOND := 41, [540].TIME.MICROSECOND := 599935, [540].EVENT := '2016/08/29   13:43:41   USER : PPS RESET FAULT BUTTON PRESSED', [541].TIME.YEAR := 2016, [541].TIME.MONTH := 8, [541].TIME.DAY := 29, [541].TIME.HOUR := 13, [541].TIME.MINUTE := 54, [541].TIME.SECOND := 27, [541].TIME.MICROSECOND := 399503, [541].EVENT := '2016/08/29   13:54:27   USER : PPS RESET FAULT BUTTON PRESSED', [542].TIME.YEAR := 2016, [542].TIME.MONTH := 8, [542].TIME.DAY := 29, [542].TIME.HOUR := 14, [542].TIME.MINUTE := 6, [542].TIME.SECOND := 43, [542].TIME.MICROSECOND := 899509, [542].EVENT := '2016/08/29   14:06:43   USER : PPS RESET FAULT BUTTON PRESSED', [543].TIME.YEAR := 2016, [543].TIME.MONTH := 8, [543].TIME.DAY := 29, [543].TIME.HOUR := 14,
        [543].TIME.MINUTE := 48, [543].TIME.SECOND := 54, [543].TIME.MICROSECOND := 799504, [543].EVENT := '2016/08/29   14:48:54   USER : PPS RESET FAULT BUTTON PRESSED', [544].TIME.YEAR := 2016, [544].TIME.MONTH := 8, [544].TIME.DAY := 29, [544].TIME.HOUR := 15, [544].TIME.MINUTE := 9, [544].TIME.SECOND := 32, [544].TIME.MICROSECOND := 399509, [544].EVENT := '2016/08/29   15:09:32   USER : PPS RESET FAULT BUTTON PRESSED', [545].TIME.YEAR := 2016, [545].TIME.MONTH := 8, [545].TIME.DAY := 29, [545].TIME.HOUR := 16, [545].TIME.SECOND := 3, [545].TIME.MICROSECOND := 899527, [545].EVENT := '2016/08/29   16:00:03   USER : PPS RESET FAULT BUTTON PRESSED', [546].TIME.YEAR := 2016, [546].TIME.MONTH := 8, [546].TIME.DAY := 29, [546].TIME.HOUR := 16, [546].TIME.MINUTE := 5, [546].TIME.SECOND := 12, [546].TIME.MICROSECOND := 399518, [546].EVENT := '2016/08/29   16:05:12   USER : PPS RESET FAULT BUTTON PRESSED', [547].TIME.YEAR := 2016, [547].TIME.MONTH := 8, [547].TIME.DAY := 29, [547].TIME.HOUR := 18, [547].TIME.MINUTE := 4, [547].TIME.SECOND := 44, [547].TIME.MICROSECOND := 499939, [547].EVENT := '2016/08/29   18:04:44   USER : PPS RESET FAULT BUTTON PRESSED', [548].TIME.YEAR := 2016, [548].TIME.MONTH := 8, [548].TIME.DAY := 29, [548].TIME.HOUR := 18, [548].TIME.MINUTE := 6, [548].TIME.SECOND := 28, [548].TIME.MICROSECOND := 799510, [548].EVENT := '2016/08/29   18:06:28   USER : PPS RESET FAULT BUTTON PRESSED', [549].TIME.YEAR := 2016, [549].TIME.MONTH := 8, [549].TIME.DAY := 30, [549].TIME.MINUTE := 17, [549].TIME.SECOND := 10, [549].TIME.MICROSECOND := 499508, [549].EVENT := '2016/08/30   00:17:10   USER : PPS RESET FAULT BUTTON PRESSED', [550].TIME.YEAR := 2016, [550].TIME.MONTH := 8, [550].TIME.DAY := 30, [550].TIME.MINUTE := 22, [550].TIME.SECOND := 48, [550].TIME.MICROSECOND := 199566, [550].EVENT := '2016/08/30   00:22:48   USER : PPS RESET FAULT BUTTON PRESSED', [551].TIME.YEAR := 2016, [551].TIME.MONTH := 8, [551].TIME.DAY := 30,
        [551].TIME.HOUR := 1, [551].TIME.MINUTE := 18, [551].TIME.SECOND := 28, [551].TIME.MICROSECOND := 399521, [551].EVENT := '2016/08/30   01:18:28   USER : PPS RESET FAULT BUTTON PRESSED', [552].TIME.YEAR := 2016, [552].TIME.MONTH := 8, [552].TIME.DAY := 30, [552].TIME.HOUR := 1, [552].TIME.MINUTE := 26, [552].TIME.SECOND := 51, [552].TIME.MICROSECOND := 499462, [552].EVENT := '2016/08/30   01:26:51   FAULT : QOW1 : Charge Outside Window Detected', [553].TIME.YEAR := 2016, [553].TIME.MONTH := 8, [553].TIME.DAY := 30, [553].TIME.HOUR := 1, [553].TIME.MINUTE := 27, [553].TIME.SECOND := 46, [553].TIME.MICROSECOND := 499506, [553].EVENT := '2016/08/30   01:27:46   USER : PPS RESET FAULT BUTTON PRESSED', [554].TIME.YEAR := 2016, [554].TIME.MONTH := 8, [554].TIME.DAY := 30, [554].TIME.HOUR := 1, [554].TIME.MINUTE := 36, [554].TIME.SECOND := 52, [554].TIME.MICROSECOND := 99482, [554].EVENT := '2016/08/30   01:36:52   FAULT : QOW1 : Charge Outside Window Detected', [555].TIME.YEAR := 2016, [555].TIME.MONTH := 8, [555].TIME.DAY := 30, [555].TIME.HOUR := 1, [555].TIME.MINUTE := 40, [555].TIME.SECOND := 49, [555].TIME.MICROSECOND := 399942, [555].EVENT := '2016/08/30   01:40:49   USER : PPS RESET FAULT BUTTON PRESSED', [556].TIME.YEAR := 2016, [556].TIME.MONTH := 8, [556].TIME.DAY := 30, [556].TIME.HOUR := 1, [556].TIME.MINUTE := 44, [556].TIME.SECOND := 19, [556].TIME.MICROSECOND := 599465, [556].EVENT := '2016/08/30   01:44:19   FAULT : QOW1 : Charge Outside Window Detected', [557].TIME.YEAR := 2016, [557].TIME.MONTH := 8, [557].TIME.DAY := 30, [557].TIME.HOUR := 1, [557].TIME.MINUTE := 45, [557].TIME.SECOND := 7, [557].TIME.MICROSECOND := 799513, [557].EVENT := '2016/08/30   01:45:07   USER : PPS RESET FAULT BUTTON PRESSED', [558].TIME.YEAR := 2016, [558].TIME.MONTH := 8, [558].TIME.DAY := 30, [558].TIME.HOUR := 2, [558].TIME.MINUTE := 54, [558].TIME.SECOND := 51, [558].TIME.MICROSECOND := 200024,
        [558].EVENT := '2016/08/30   02:54:51   USER : PPS RESET FAULT BUTTON PRESSED', [559].TIME.YEAR := 2016, [559].TIME.MONTH := 8, [559].TIME.DAY := 30, [559].TIME.HOUR := 4, [559].TIME.SECOND := 16, [559].TIME.MICROSECOND := 199465, [559].EVENT := '2016/08/30   04:00:16   FAULT : QOW1 : Charge Outside Window Detected', [560].TIME.YEAR := 2016, [560].TIME.MONTH := 8, [560].TIME.DAY := 30, [560].TIME.HOUR := 4, [560].TIME.MINUTE := 9, [560].TIME.SECOND := 53, [560].TIME.MICROSECOND := 599547, [560].EVENT := '2016/08/30   04:09:53   USER : PPS RESET FAULT BUTTON PRESSED', [561].TIME.YEAR := 2016, [561].TIME.MONTH := 8, [561].TIME.DAY := 30, [561].TIME.HOUR := 4, [561].TIME.MINUTE := 10, [561].TIME.SECOND := 40, [561].TIME.MICROSECOND := 699561, [561].EVENT := '2016/08/30   04:10:40   USER : PPS RESET FAULT BUTTON PRESSED', [562].TIME.YEAR := 2016, [562].TIME.MONTH := 8, [562].TIME.DAY := 31, [562].TIME.HOUR := 9, [562].TIME.MINUTE := 16, [562].TIME.SECOND := 39, [562].TIME.MICROSECOND := 299549, [562].EVENT := '2016/08/31   09:16:39   USER : PPS RESET FAULT BUTTON PRESSED', [563].TIME.YEAR := 2016, [563].TIME.MONTH := 8, [563].TIME.DAY := 31, [563].TIME.HOUR := 9, [563].TIME.MINUTE := 16, [563].TIME.SECOND := 39, [563].TIME.MICROSECOND := 699506, [563].EVENT := '2016/08/31   09:16:39   USER : PPS RESET FAULT BUTTON PRESSED', [564].TIME.YEAR := 2016, [564].TIME.MONTH := 8, [564].TIME.DAY := 31, [564].TIME.HOUR := 9, [564].TIME.MINUTE := 22, [564].TIME.SECOND := 24, [564].TIME.MICROSECOND := 899509, [564].EVENT := '2016/08/31   09:22:24   USER : PPS RESET FAULT BUTTON PRESSED', [565].TIME.YEAR := 2016, [565].TIME.MONTH := 8, [565].TIME.DAY := 31, [565].TIME.HOUR := 9, [565].TIME.MINUTE := 32, [565].TIME.SECOND := 38, [565].TIME.MICROSECOND := 999507, [565].EVENT := '2016/08/31   09:32:38   USER : PPS RESET FAULT BUTTON PRESSED', [566].TIME.YEAR := 2016, [566].TIME.MONTH := 8, [566].TIME.DAY := 31, [566].TIME.HOUR := 9,
        [566].TIME.MINUTE := 38, [566].TIME.SECOND := 34, [566].TIME.MICROSECOND := 599506, [566].EVENT := '2016/08/31   09:38:34   USER : PPS RESET FAULT BUTTON PRESSED', [567].TIME.YEAR := 2016, [567].TIME.MONTH := 8, [567].TIME.DAY := 31, [567].TIME.HOUR := 10, [567].TIME.MINUTE := 12, [567].TIME.SECOND := 30, [567].TIME.MICROSECOND := 399465, [567].EVENT := '2016/08/31   10:12:30   FAULT : QOW1 : Charge Outside Window Detected', [568].TIME.YEAR := 2016, [568].TIME.MONTH := 8, [568].TIME.DAY := 31, [568].TIME.HOUR := 10, [568].TIME.MINUTE := 21, [568].TIME.SECOND := 36, [568].TIME.MICROSECOND := 499494, [568].EVENT := '2016/08/31   10:21:36   USER : RESET FAULT BUTTON PRESSED', [569].TIME.YEAR := 2016, [569].TIME.MONTH := 8, [569].TIME.DAY := 31, [569].TIME.HOUR := 10, [569].TIME.MINUTE := 28, [569].TIME.SECOND := 35, [569].TIME.MICROSECOND := 499465, [569].EVENT := '2016/08/31   10:28:35   FAULT : QOW1 : Charge Outside Window Detected', [570].TIME.YEAR := 2016, [570].TIME.MONTH := 8, [570].TIME.DAY := 31, [570].TIME.HOUR := 10, [570].TIME.MINUTE := 33, [570].TIME.SECOND := 22, [570].TIME.MICROSECOND := 199502, [570].EVENT := '2016/08/31   10:33:22   USER : RESET FAULT BUTTON PRESSED', [571].TIME.YEAR := 2016, [571].TIME.MONTH := 8, [571].TIME.DAY := 31, [571].TIME.HOUR := 10, [571].TIME.MINUTE := 56, [571].TIME.SECOND := 40, [571].TIME.MICROSECOND := 999510, [571].EVENT := '2016/08/31   10:56:40   USER : PPS RESET FAULT BUTTON PRESSED', [572].TIME.YEAR := 2016, [572].TIME.MONTH := 8, [572].TIME.DAY := 31, [572].TIME.HOUR := 14, [572].TIME.MINUTE := 58, [572].TIME.SECOND := 51, [572].TIME.MICROSECOND := 999554, [572].EVENT := '2016/08/31   14:58:51   USER : PPS RESET FAULT BUTTON PRESSED', [573].TIME.YEAR := 2016, [573].TIME.MONTH := 8, [573].TIME.DAY := 31, [573].TIME.HOUR := 15, [573].TIME.SECOND := 21, [573].TIME.MICROSECOND := 300122, [573].EVENT := '2016/08/31   15:00:21   USER : PPS RESET FAULT BUTTON PRESSED', [574].TIME.YEAR := 2016,
        [574].TIME.MONTH := 8, [574].TIME.DAY := 31, [574].TIME.HOUR := 15, [574].TIME.SECOND := 21, [574].TIME.MICROSECOND := 699505, [574].EVENT := '2016/08/31   15:00:21   USER : PPS RESET FAULT BUTTON PRESSED', [575].TIME.YEAR := 2016, [575].TIME.MONTH := 8, [575].TIME.DAY := 31, [575].TIME.HOUR := 15, [575].TIME.SECOND := 21, [575].TIME.MICROSECOND := 999507, [575].EVENT := '2016/08/31   15:00:21   USER : PPS RESET FAULT BUTTON PRESSED', [576].TIME.YEAR := 2016, [576].TIME.MONTH := 8, [576].TIME.DAY := 31, [576].TIME.HOUR := 15, [576].TIME.SECOND := 22, [576].TIME.MICROSECOND := 199505, [576].EVENT := '2016/08/31   15:00:22   USER : PPS RESET FAULT BUTTON PRESSED', [577].TIME.YEAR := 2016, [577].TIME.MONTH := 8, [577].TIME.DAY := 31, [577].TIME.HOUR := 15, [577].TIME.SECOND := 22, [577].TIME.MICROSECOND := 499515, [577].EVENT := '2016/08/31   15:00:22   USER : PPS RESET FAULT BUTTON PRESSED', [578].TIME.YEAR := 2016, [578].TIME.MONTH := 8, [578].TIME.DAY := 31, [578].TIME.HOUR := 15, [578].TIME.SECOND := 22, [578].TIME.MICROSECOND := 799935, [578].EVENT := '2016/08/31   15:00:22   USER : PPS RESET FAULT BUTTON PRESSED', [579].TIME.YEAR := 2016, [579].TIME.MONTH := 8, [579].TIME.DAY := 31, [579].TIME.HOUR := 15, [579].TIME.SECOND := 23, [579].TIME.MICROSECOND := 99558, [579].EVENT := '2016/08/31   15:00:23   USER : PPS RESET FAULT BUTTON PRESSED', [580].TIME.YEAR := 2016, [580].TIME.MONTH := 8, [580].TIME.DAY := 31, [580].TIME.HOUR := 15, [580].TIME.SECOND := 43, [580].TIME.MICROSECOND := 199938, [580].EVENT := '2016/08/31   15:00:43   USER : PPS RESET FAULT BUTTON PRESSED', [581].TIME.YEAR := 2016, [581].TIME.MONTH := 8, [581].TIME.DAY := 31, [581].TIME.HOUR := 15, [581].TIME.MINUTE := 15, [581].TIME.SECOND := 47, [581].TIME.MICROSECOND := 499512, [581].EVENT := '2016/08/31   15:15:47   USER : PPS RESET FAULT BUTTON PRESSED', [582].TIME.YEAR := 2016, [582].TIME.MONTH := 8, [582].TIME.DAY := 31, [582].TIME.HOUR := 15,
        [582].TIME.MINUTE := 17, [582].TIME.SECOND := 1, [582].TIME.MICROSECOND := 300023, [582].EVENT := '2016/08/31   15:17:01   USER : PPS RESET FAULT BUTTON PRESSED', [583].TIME.YEAR := 2016, [583].TIME.MONTH := 8, [583].TIME.DAY := 31, [583].TIME.HOUR := 15, [583].TIME.MINUTE := 17, [583].TIME.SECOND := 2, [583].TIME.MICROSECOND := 899511, [583].EVENT := '2016/08/31   15:17:02   USER : PPS RESET FAULT BUTTON PRESSED', [584].TIME.YEAR := 2016, [584].TIME.MONTH := 8, [584].TIME.DAY := 31, [584].TIME.HOUR := 15, [584].TIME.MINUTE := 21, [584].TIME.SECOND := 1, [584].TIME.MICROSECOND := 300025, [584].EVENT := '2016/08/31   15:21:01   USER : PPS RESET FAULT BUTTON PRESSED', [585].TIME.YEAR := 2016, [585].TIME.MONTH := 8, [585].TIME.DAY := 31, [585].TIME.HOUR := 15, [585].TIME.MINUTE := 30, [585].TIME.SECOND := 24, [585].TIME.MICROSECOND := 599509, [585].EVENT := '2016/08/31   15:30:24   USER : PPS RESET FAULT BUTTON PRESSED', [586].TIME.YEAR := 2016, [586].TIME.MONTH := 8, [586].TIME.DAY := 31, [586].TIME.HOUR := 15, [586].TIME.MINUTE := 30, [586].TIME.SECOND := 28, [586].TIME.MICROSECOND := 399520, [586].EVENT := '2016/08/31   15:30:28   USER : PPS RESET FAULT BUTTON PRESSED', [587].TIME.YEAR := 2016, [587].TIME.MONTH := 8, [587].TIME.DAY := 31, [587].TIME.HOUR := 15, [587].TIME.MINUTE := 30, [587].TIME.SECOND := 30, [587].TIME.MICROSECOND := 699530, [587].EVENT := '2016/08/31   15:30:30   USER : PPS RESET FAULT BUTTON PRESSED', [588].TIME.YEAR := 2016, [588].TIME.MONTH := 8, [588].TIME.DAY := 31, [588].TIME.HOUR := 15, [588].TIME.MINUTE := 30, [588].TIME.SECOND := 45, [588].TIME.MICROSECOND := 499516, [588].EVENT := '2016/08/31   15:30:45   USER : PPS RESET FAULT BUTTON PRESSED', [589].TIME.YEAR := 2016, [589].TIME.MONTH := 8, [589].TIME.DAY := 31, [589].TIME.HOUR := 15, [589].TIME.MINUTE := 30, [589].TIME.SECOND := 46, [589].TIME.MICROSECOND := 899506, [589].EVENT := '2016/08/31   15:30:46   USER : PPS RESET FAULT BUTTON PRESSED',
        [590].TIME.YEAR := 2016, [590].TIME.MONTH := 8, [590].TIME.DAY := 31, [590].TIME.HOUR := 15, [590].TIME.MINUTE := 30, [590].TIME.SECOND := 47, [590].TIME.MICROSECOND := 99939, [590].EVENT := '2016/08/31   15:30:47   USER : PPS RESET FAULT BUTTON PRESSED', [591].TIME.YEAR := 2016, [591].TIME.MONTH := 8, [591].TIME.DAY := 31, [591].TIME.HOUR := 15, [591].TIME.MINUTE := 30, [591].TIME.SECOND := 47, [591].TIME.MICROSECOND := 299504, [591].EVENT := '2016/08/31   15:30:47   USER : PPS RESET FAULT BUTTON PRESSED', [592].TIME.YEAR := 2016, [592].TIME.MONTH := 8, [592].TIME.DAY := 31, [592].TIME.HOUR := 15, [592].TIME.MINUTE := 30, [592].TIME.SECOND := 47, [592].TIME.MICROSECOND := 499507, [592].EVENT := '2016/08/31   15:30:47   USER : PPS RESET FAULT BUTTON PRESSED', [593].TIME.YEAR := 2016, [593].TIME.MONTH := 8, [593].TIME.DAY := 31, [593].TIME.HOUR := 15, [593].TIME.MINUTE := 30, [593].TIME.SECOND := 47, [593].TIME.MICROSECOND := 699508, [593].EVENT := '2016/08/31   15:30:47   USER : PPS RESET FAULT BUTTON PRESSED', [594].TIME.YEAR := 2016, [594].TIME.MONTH := 8, [594].TIME.DAY := 31, [594].TIME.HOUR := 15, [594].TIME.MINUTE := 40, [594].TIME.SECOND := 56, [594].TIME.MICROSECOND := 99510, [594].EVENT := '2016/08/31   15:40:56   USER : PPS RESET FAULT BUTTON PRESSED', [595].TIME.YEAR := 2016, [595].TIME.MONTH := 8, [595].TIME.DAY := 31, [595].TIME.HOUR := 15, [595].TIME.MINUTE := 41, [595].TIME.MICROSECOND := 399504, [595].EVENT := '2016/08/31   15:41:00   USER : PPS RESET FAULT BUTTON PRESSED', [596].TIME.YEAR := 2016, [596].TIME.MONTH := 8, [596].TIME.DAY := 31, [596].TIME.HOUR := 15, [596].TIME.MINUTE := 42, [596].TIME.SECOND := 55, [596].TIME.MICROSECOND := 899521, [596].EVENT := '2016/08/31   15:42:55   USER : PPS RESET FAULT BUTTON PRESSED', [597].TIME.YEAR := 2016, [597].TIME.MONTH := 8, [597].TIME.DAY := 31, [597].TIME.HOUR := 15, [597].TIME.MINUTE := 44,
        [597].TIME.SECOND := 7, [597].TIME.MICROSECOND := 299608, [597].EVENT := '2016/08/31   15:44:07   FAULT : QOW1 : Charge Outside Window Detected', [598].TIME.YEAR := 2016, [598].TIME.MONTH := 8, [598].TIME.DAY := 31, [598].TIME.HOUR := 15, [598].TIME.MINUTE := 44, [598].TIME.SECOND := 42, [598].TIME.MICROSECOND := 899581, [598].EVENT := '2016/08/31   15:44:42   USER : RESET FAULT BUTTON PRESSED', [599].TIME.YEAR := 2016, [599].TIME.MONTH := 8, [599].TIME.DAY := 31, [599].TIME.HOUR := 15, [599].TIME.MINUTE := 46, [599].TIME.SECOND := 43, [599].TIME.MICROSECOND := 299978, [599].EVENT := '2016/08/31   15:46:43   FAULT : QOW1 : Charge Outside Window Detected', [600].TIME.YEAR := 2016, [600].TIME.MONTH := 8, [600].TIME.DAY := 31, [600].TIME.HOUR := 15, [600].TIME.MINUTE := 46, [600].TIME.SECOND := 43, [600].TIME.MICROSECOND := 599511, [600].EVENT := '2016/08/31   15:46:43   USER : PPS RESET FAULT BUTTON PRESSED', [601].TIME.YEAR := 2016, [601].TIME.MONTH := 8, [601].TIME.DAY := 31, [601].TIME.HOUR := 15, [601].TIME.MINUTE := 46, [601].TIME.SECOND := 53, [601].TIME.MICROSECOND := 799490, [601].EVENT := '2016/08/31   15:46:53   USER : RESET FAULT BUTTON PRESSED', [602].TIME.YEAR := 2016, [602].TIME.MONTH := 8, [602].TIME.DAY := 31, [602].TIME.HOUR := 15, [602].TIME.MINUTE := 46, [602].TIME.SECOND := 54, [602].TIME.MICROSECOND := 399654, [602].EVENT := '2016/08/31   15:46:54   USER : PPS RESET FAULT BUTTON PRESSED', [603].TIME.YEAR := 2016, [603].TIME.MONTH := 8, [603].TIME.DAY := 31, [603].TIME.HOUR := 15, [603].TIME.MINUTE := 47, [603].TIME.SECOND := 33, [603].TIME.MICROSECOND := 699510, [603].EVENT := '2016/08/31   15:47:33   USER : PPS RESET FAULT BUTTON PRESSED', [604].TIME.YEAR := 2016, [604].TIME.MONTH := 8, [604].TIME.DAY := 31, [604].TIME.HOUR := 15, [604].TIME.MINUTE := 47, [604].TIME.SECOND := 34, [604].TIME.MICROSECOND := 499721, [604].EVENT := '2016/08/31   15:47:34   USER : PPS RESET FAULT BUTTON PRESSED', [605].TIME.YEAR := 2016,
        [605].TIME.MONTH := 8, [605].TIME.DAY := 31, [605].TIME.HOUR := 15, [605].TIME.MINUTE := 47, [605].TIME.SECOND := 34, [605].TIME.MICROSECOND := 999510, [605].EVENT := '2016/08/31   15:47:34   USER : PPS RESET FAULT BUTTON PRESSED', [606].TIME.YEAR := 2016, [606].TIME.MONTH := 8, [606].TIME.DAY := 31, [606].TIME.HOUR := 15, [606].TIME.MINUTE := 47, [606].TIME.SECOND := 35, [606].TIME.MICROSECOND := 199521, [606].EVENT := '2016/08/31   15:47:35   USER : PPS RESET FAULT BUTTON PRESSED', [607].TIME.YEAR := 2016, [607].TIME.MONTH := 8, [607].TIME.DAY := 31, [607].TIME.HOUR := 15, [607].TIME.MINUTE := 47, [607].TIME.SECOND := 35, [607].TIME.MICROSECOND := 399505, [607].EVENT := '2016/08/31   15:47:35   USER : PPS RESET FAULT BUTTON PRESSED', [608].TIME.YEAR := 2016, [608].TIME.MONTH := 8, [608].TIME.DAY := 31, [608].TIME.HOUR := 15, [608].TIME.MINUTE := 47, [608].TIME.SECOND := 35, [608].TIME.MICROSECOND := 699524, [608].EVENT := '2016/08/31   15:47:35   USER : PPS RESET FAULT BUTTON PRESSED', [609].TIME.YEAR := 2016, [609].TIME.MONTH := 8, [609].TIME.DAY := 31, [609].TIME.HOUR := 15, [609].TIME.MINUTE := 47, [609].TIME.SECOND := 35, [609].TIME.MICROSECOND := 899505, [609].EVENT := '2016/08/31   15:47:35   USER : PPS RESET FAULT BUTTON PRESSED', [610].TIME.YEAR := 2016, [610].TIME.MONTH := 8, [610].TIME.DAY := 31, [610].TIME.HOUR := 15, [610].TIME.MINUTE := 47, [610].TIME.SECOND := 36, [610].TIME.MICROSECOND := 99517, [610].EVENT := '2016/08/31   15:47:36   USER : PPS RESET FAULT BUTTON PRESSED', [611].TIME.YEAR := 2016, [611].TIME.MONTH := 8, [611].TIME.DAY := 31, [611].TIME.HOUR := 15, [611].TIME.MINUTE := 47, [611].TIME.SECOND := 36, [611].TIME.MICROSECOND := 800018, [611].EVENT := '2016/08/31   15:47:36   USER : PPS RESET FAULT BUTTON PRESSED', [612].TIME.YEAR := 2016, [612].TIME.MONTH := 8, [612].TIME.DAY := 31, [612].TIME.HOUR := 15, [612].TIME.MINUTE := 47,
        [612].TIME.SECOND := 36, [612].TIME.MICROSECOND := 999505, [612].EVENT := '2016/08/31   15:47:36   USER : PPS RESET FAULT BUTTON PRESSED', [613].TIME.YEAR := 2016, [613].TIME.MONTH := 8, [613].TIME.DAY := 31, [613].TIME.HOUR := 15, [613].TIME.MINUTE := 47, [613].TIME.SECOND := 37, [613].TIME.MICROSECOND := 499504, [613].EVENT := '2016/08/31   15:47:37   USER : PPS RESET FAULT BUTTON PRESSED', [614].TIME.YEAR := 2016, [614].TIME.MONTH := 8, [614].TIME.DAY := 31, [614].TIME.HOUR := 15, [614].TIME.MINUTE := 47, [614].TIME.SECOND := 37, [614].TIME.MICROSECOND := 999553, [614].EVENT := '2016/08/31   15:47:37   USER : PPS RESET FAULT BUTTON PRESSED', [615].TIME.YEAR := 2016, [615].TIME.MONTH := 8, [615].TIME.DAY := 31, [615].TIME.HOUR := 15, [615].TIME.MINUTE := 47, [615].TIME.SECOND := 38, [615].TIME.MICROSECOND := 199505, [615].EVENT := '2016/08/31   15:47:38   USER : PPS RESET FAULT BUTTON PRESSED', [616].TIME.YEAR := 2016, [616].TIME.MONTH := 8, [616].TIME.DAY := 31, [616].TIME.HOUR := 15, [616].TIME.MINUTE := 47, [616].TIME.SECOND := 38, [616].TIME.MICROSECOND := 499513, [616].EVENT := '2016/08/31   15:47:38   USER : PPS RESET FAULT BUTTON PRESSED', [617].TIME.YEAR := 2016, [617].TIME.MONTH := 8, [617].TIME.DAY := 31, [617].TIME.HOUR := 15, [617].TIME.MINUTE := 47, [617].TIME.SECOND := 38, [617].TIME.MICROSECOND := 999515, [617].EVENT := '2016/08/31   15:47:38   USER : PPS RESET FAULT BUTTON PRESSED', [618].TIME.YEAR := 2016, [618].TIME.MONTH := 8, [618].TIME.DAY := 31, [618].TIME.HOUR := 15, [618].TIME.MINUTE := 48, [618].TIME.SECOND := 45, [618].TIME.MICROSECOND := 99936, [618].EVENT := '2016/08/31   15:48:45   USER : PPS RESET FAULT BUTTON PRESSED', [619].TIME.YEAR := 2016, [619].TIME.MONTH := 8, [619].TIME.DAY := 31, [619].TIME.HOUR := 15, [619].TIME.MINUTE := 48, [619].TIME.SECOND := 45, [619].TIME.MICROSECOND := 600028, [619].EVENT := '2016/08/31   15:48:45   USER : PPS RESET FAULT BUTTON PRESSED', [620].TIME.YEAR := 2016,
        [620].TIME.MONTH := 8, [620].TIME.DAY := 31, [620].TIME.HOUR := 15, [620].TIME.MINUTE := 50, [620].TIME.SECOND := 55, [620].TIME.MICROSECOND := 299465, [620].EVENT := '2016/08/31   15:50:55   FAULT : QOW1 : Charge Outside Window Detected', [621].TIME.YEAR := 2016, [621].TIME.MONTH := 8, [621].TIME.DAY := 31, [621].TIME.HOUR := 15, [621].TIME.MINUTE := 51, [621].TIME.SECOND := 13, [621].TIME.MICROSECOND := 699495, [621].EVENT := '2016/08/31   15:51:13   USER : RESET FAULT BUTTON PRESSED', [622].TIME.YEAR := 2016, [622].TIME.MONTH := 8, [622].TIME.DAY := 31, [622].TIME.HOUR := 15, [622].TIME.MINUTE := 51, [622].TIME.SECOND := 20, [622].TIME.MICROSECOND := 799509, [622].EVENT := '2016/08/31   15:51:20   USER : PPS RESET FAULT BUTTON PRESSED', [623].TIME.YEAR := 2016, [623].TIME.MONTH := 8, [623].TIME.DAY := 31, [623].TIME.HOUR := 15, [623].TIME.MINUTE := 51, [623].TIME.SECOND := 23, [623].TIME.MICROSECOND := 23, [623].EVENT := '2016/08/31   15:51:23   USER : PPS RESET FAULT BUTTON PRESSED', [624].TIME.YEAR := 2016, [624].TIME.MONTH := 8, [624].TIME.DAY := 31, [624].TIME.HOUR := 15, [624].TIME.MINUTE := 54, [624].TIME.SECOND := 35, [624].TIME.MICROSECOND := 799458, [624].EVENT := '2016/08/31   15:54:35   FAULT : QOW1 : Charge Outside Window Detected', [625].TIME.YEAR := 2016, [625].TIME.MONTH := 8, [625].TIME.DAY := 31, [625].TIME.HOUR := 15, [625].TIME.MINUTE := 54, [625].TIME.SECOND := 36, [625].TIME.MICROSECOND := 199508, [625].EVENT := '2016/08/31   15:54:36   USER : PPS RESET FAULT BUTTON PRESSED', [626].TIME.YEAR := 2016, [626].TIME.MONTH := 8, [626].TIME.DAY := 31, [626].TIME.HOUR := 15, [626].TIME.MINUTE := 54, [626].TIME.SECOND := 42, [626].TIME.MICROSECOND := 99634, [626].EVENT := '2016/08/31   15:54:42   USER : RESET FAULT BUTTON PRESSED', [627].TIME.YEAR := 2016, [627].TIME.MONTH := 8, [627].TIME.DAY := 31, [627].TIME.HOUR := 16, [627].TIME.MINUTE := 2,
        [627].TIME.SECOND := 37, [627].TIME.MICROSECOND := 25, [627].EVENT := '2016/08/31   16:02:37   USER : PPS RESET FAULT BUTTON PRESSED', [628].TIME.YEAR := 2016, [628].TIME.MONTH := 9, [628].TIME.DAY := 1, [628].TIME.HOUR := 9, [628].TIME.MINUTE := 30, [628].TIME.SECOND := 5, [628].TIME.MICROSECOND := 399505, [628].EVENT := '2016/09/01   09:30:05   USER : PPS RESET FAULT BUTTON PRESSED', [629].TIME.YEAR := 2016, [629].TIME.MONTH := 9, [629].TIME.DAY := 1, [629].TIME.HOUR := 9, [629].TIME.MINUTE := 43, [629].TIME.SECOND := 2, [629].TIME.MICROSECOND := 299464, [629].EVENT := '2016/09/01   09:43:02   FAULT : QOW1 : Charge Outside Window Detected', [630].TIME.YEAR := 2016, [630].TIME.MONTH := 9, [630].TIME.DAY := 1, [630].TIME.HOUR := 9, [630].TIME.MINUTE := 43, [630].TIME.SECOND := 51, [630].TIME.MICROSECOND := 299492, [630].EVENT := '2016/09/01   09:43:51   USER : RESET FAULT BUTTON PRESSED', [631].TIME.YEAR := 2016, [631].TIME.MONTH := 9, [631].TIME.DAY := 1, [631].TIME.HOUR := 9, [631].TIME.MINUTE := 45, [631].TIME.SECOND := 32, [631].TIME.MICROSECOND := 899523, [631].EVENT := '2016/09/01   09:45:32   USER : PPS RESET FAULT BUTTON PRESSED', [632].TIME.YEAR := 2016, [632].TIME.MONTH := 9, [632].TIME.DAY := 1, [632].TIME.HOUR := 9, [632].TIME.MINUTE := 47, [632].TIME.SECOND := 2, [632].TIME.MICROSECOND := 399504, [632].EVENT := '2016/09/01   09:47:02   USER : PPS RESET FAULT BUTTON PRESSED', [633].TIME.YEAR := 2016, [633].TIME.MONTH := 9, [633].TIME.DAY := 1, [633].TIME.HOUR := 9, [633].TIME.MINUTE := 52, [633].TIME.SECOND := 45, [633].TIME.MICROSECOND := 99508, [633].EVENT := '2016/09/01   09:52:45   USER : PPS RESET FAULT BUTTON PRESSED', [634].TIME.YEAR := 2016, [634].TIME.MONTH := 9, [634].TIME.DAY := 1, [634].TIME.HOUR := 9, [634].TIME.MINUTE := 54, [634].TIME.SECOND := 17, [634].TIME.MICROSECOND := 599511, [634].EVENT := '2016/09/01   09:54:17   USER : PPS RESET FAULT BUTTON PRESSED', [635].TIME.YEAR := 2016,
        [635].TIME.MONTH := 9, [635].TIME.DAY := 1, [635].TIME.HOUR := 9, [635].TIME.MINUTE := 54, [635].TIME.SECOND := 19, [635].TIME.MICROSECOND := 300025, [635].EVENT := '2016/09/01   09:54:19   USER : PPS RESET FAULT BUTTON PRESSED', [636].TIME.YEAR := 2016, [636].TIME.MONTH := 9, [636].TIME.DAY := 1, [636].TIME.HOUR := 9, [636].TIME.MINUTE := 54, [636].TIME.SECOND := 23, [636].TIME.MICROSECOND := 199509, [636].EVENT := '2016/09/01   09:54:23   USER : PPS RESET FAULT BUTTON PRESSED', [637].TIME.YEAR := 2016, [637].TIME.MONTH := 9, [637].TIME.DAY := 1, [637].TIME.HOUR := 9, [637].TIME.MINUTE := 54, [637].TIME.SECOND := 26, [637].TIME.MICROSECOND := 599512, [637].EVENT := '2016/09/01   09:54:26   USER : PPS RESET FAULT BUTTON PRESSED', [638].TIME.YEAR := 2016, [638].TIME.MONTH := 9, [638].TIME.DAY := 1, [638].TIME.HOUR := 9, [638].TIME.MINUTE := 54, [638].TIME.SECOND := 39, [638].TIME.MICROSECOND := 399513, [638].EVENT := '2016/09/01   09:54:39   USER : PPS RESET FAULT BUTTON PRESSED', [639].TIME.YEAR := 2016, [639].TIME.MONTH := 9, [639].TIME.DAY := 1, [639].TIME.HOUR := 10, [639].TIME.MINUTE := 36, [639].TIME.SECOND := 1, [639].TIME.MICROSECOND := 499843, [639].EVENT := '2016/09/01   10:36:01   USER : PPS RESET FAULT BUTTON PRESSED', [640].TIME.YEAR := 2016, [640].TIME.MONTH := 9, [640].TIME.DAY := 12, [640].TIME.HOUR := 14, [640].TIME.MINUTE := 18, [640].TIME.SECOND := 57, [640].TIME.MICROSECOND := 899510, [640].EVENT := '2016/09/12   14:18:57   USER : PPS RESET FAULT BUTTON PRESSED', [641].TIME.YEAR := 2016, [641].TIME.MONTH := 9, [641].TIME.DAY := 12, [641].TIME.HOUR := 14, [641].TIME.MINUTE := 19, [641].TIME.SECOND := 21, [641].TIME.MICROSECOND := 799500, [641].EVENT := '2016/09/12   14:19:21   USER : PPS RESET FAULT BUTTON PRESSED', [642].TIME.YEAR := 2016, [642].TIME.MONTH := 9, [642].TIME.DAY := 12, [642].TIME.HOUR := 14, [642].TIME.MINUTE := 33,
        [642].TIME.SECOND := 20, [642].TIME.MICROSECOND := 99503, [642].EVENT := '2016/09/12   14:33:20   USER : PPS RESET FAULT BUTTON PRESSED', [643].TIME.YEAR := 2016, [643].TIME.MONTH := 9, [643].TIME.DAY := 12, [643].TIME.HOUR := 15, [643].TIME.MINUTE := 17, [643].TIME.SECOND := 46, [643].TIME.MICROSECOND := 899462, [643].EVENT := '2016/09/12   15:17:46   FAULT : QOW1 : Charge Outside Window Detected', [644].TIME.YEAR := 2016, [644].TIME.MONTH := 9, [644].TIME.DAY := 12, [644].TIME.HOUR := 15, [644].TIME.MINUTE := 17, [644].TIME.SECOND := 57, [644].TIME.MICROSECOND := 299982, [644].EVENT := '2016/09/12   15:17:57   FAULT : Self Test 2 Charge (B-A) LOW', [645].TIME.YEAR := 2016, [645].TIME.MONTH := 9, [645].TIME.DAY := 12, [645].TIME.HOUR := 15, [645].TIME.MINUTE := 18, [645].TIME.SECOND := 1, [645].TIME.MICROSECOND := 399902, [645].EVENT := '2016/09/12   15:18:01   FAULT : Self Test 2 NO QAT DETECTED', [646].TIME.YEAR := 2016, [646].TIME.MONTH := 9, [646].TIME.DAY := 12, [646].TIME.HOUR := 15, [646].TIME.MINUTE := 18, [646].TIME.SECOND := 1, [646].TIME.MICROSECOND := 899788, [646].EVENT := '2016/09/12   15:18:01   FAULT : Self Test 1 Charge (A-B) LOW', [647].TIME.YEAR := 2016, [647].TIME.MONTH := 9, [647].TIME.DAY := 12, [647].TIME.HOUR := 15, [647].TIME.MINUTE := 18, [647].TIME.SECOND := 1, [647].TIME.MICROSECOND := 900364, [647].EVENT := '2016/09/12   15:18:01   FAULT : Self Test 1 NO QAT DETECTED', [648].TIME.YEAR := 2016, [648].TIME.MONTH := 9, [648].TIME.DAY := 12, [648].TIME.HOUR := 15, [648].TIME.MINUTE := 18, [648].TIME.SECOND := 2, [648].TIME.MICROSECOND := 399803, [648].EVENT := '2016/09/12   15:18:02   FAULT : Self Test 1 Charge (B-A) LOW', [649].TIME.YEAR := 2016, [649].TIME.MONTH := 9, [649].TIME.DAY := 12, [649].TIME.HOUR := 15, [649].TIME.MINUTE := 18, [649].TIME.SECOND := 2, [649].TIME.MICROSECOND := 899892, [649].EVENT := '2016/09/12   15:18:02   FAULT : Self Test 2 Charge (A-B) LOW', [650].TIME.YEAR := 2016,
        [650].TIME.MONTH := 9, [650].TIME.DAY := 13, [650].TIME.HOUR := 9, [650].TIME.MINUTE := 7, [650].TIME.SECOND := 55, [650].TIME.MICROSECOND := 399494, [650].EVENT := '2016/09/13   09:07:55   USER : RESET FAULT BUTTON PRESSED', [651].TIME.YEAR := 2016, [651].TIME.MONTH := 9, [651].TIME.DAY := 13, [651].TIME.HOUR := 9, [651].TIME.MINUTE := 7, [651].TIME.SECOND := 55, [651].TIME.MICROSECOND := 599842, [651].EVENT := '2016/09/13   09:07:55   FAULT : Self Test 2 Charge (B-A) LOW', [652].TIME.YEAR := 2016, [652].TIME.MONTH := 9, [652].TIME.DAY := 13, [652].TIME.HOUR := 9, [652].TIME.MINUTE := 7, [652].TIME.SECOND := 55, [652].TIME.MICROSECOND := 600404, [652].EVENT := '2016/09/13   09:07:55   FAULT : Self Test 2 NO QAT DETECTED', [653].TIME.YEAR := 2016, [653].TIME.MONTH := 9, [653].TIME.DAY := 13, [653].TIME.HOUR := 9, [653].TIME.MINUTE := 7, [653].TIME.SECOND := 56, [653].TIME.MICROSECOND := 99781, [653].EVENT := '2016/09/13   09:07:56   FAULT : Self Test 1 Charge (A-B) LOW', [654].TIME.YEAR := 2016, [654].TIME.MONTH := 9, [654].TIME.DAY := 13, [654].TIME.HOUR := 9, [654].TIME.MINUTE := 7, [654].TIME.SECOND := 56, [654].TIME.MICROSECOND := 100359, [654].EVENT := '2016/09/13   09:07:56   FAULT : Self Test 1 NO QAT DETECTED', [655].TIME.YEAR := 2016, [655].TIME.MONTH := 9, [655].TIME.DAY := 13, [655].TIME.HOUR := 9, [655].TIME.MINUTE := 7, [655].TIME.SECOND := 56, [655].TIME.MICROSECOND := 599794, [655].EVENT := '2016/09/13   09:07:56   FAULT : Self Test 1 Charge (B-A) LOW', [656].TIME.YEAR := 2016, [656].TIME.MONTH := 9, [656].TIME.DAY := 13, [656].TIME.HOUR := 9, [656].TIME.MINUTE := 7, [656].TIME.SECOND := 57, [656].TIME.MICROSECOND := 199832, [656].EVENT := '2016/09/13   09:07:57   FAULT : Self Test 2 Charge (A-B) LOW', [657].TIME.YEAR := 2016, [657].TIME.MONTH := 9, [657].TIME.DAY := 13, [657].TIME.HOUR := 9, [657].TIME.MINUTE := 7,
        [657].TIME.SECOND := 59, [657].TIME.MICROSECOND := 200155, [657].EVENT := '2016/09/13   09:07:59   FAULT : Self Test 2 Charge (A-B) LOW', [658].TIME.YEAR := 2016, [658].TIME.MONTH := 9, [658].TIME.DAY := 13, [658].TIME.HOUR := 9, [658].TIME.MINUTE := 7, [658].TIME.SECOND := 59, [658].TIME.MICROSECOND := 200676, [658].EVENT := '2016/09/13   09:07:59   FAULT : Self Test 2 NO QAT DETECTED', [659].TIME.YEAR := 2016, [659].TIME.MONTH := 9, [659].TIME.DAY := 13, [659].TIME.HOUR := 9, [659].TIME.MINUTE := 7, [659].TIME.SECOND := 59, [659].TIME.MICROSECOND := 399492, [659].EVENT := '2016/09/13   09:07:59   USER : RESET FAULT BUTTON PRESSED', [660].TIME.YEAR := 2016, [660].TIME.MONTH := 9, [660].TIME.DAY := 13, [660].TIME.HOUR := 9, [660].TIME.MINUTE := 7, [660].TIME.SECOND := 59, [660].TIME.MICROSECOND := 699901, [660].EVENT := '2016/09/13   09:07:59   FAULT : Self Test 2 Charge (B-A) LOW', [661].TIME.YEAR := 2016, [661].TIME.MONTH := 9, [661].TIME.DAY := 13, [661].TIME.HOUR := 9, [661].TIME.MINUTE := 8, [661].TIME.MICROSECOND := 199770, [661].EVENT := '2016/09/13   09:08:00   FAULT : Self Test 1 Charge (A-B) LOW', [662].TIME.YEAR := 2016, [662].TIME.MONTH := 9, [662].TIME.DAY := 13, [662].TIME.HOUR := 9, [662].TIME.MINUTE := 8, [662].TIME.MICROSECOND := 200347, [662].EVENT := '2016/09/13   09:08:00   FAULT : Self Test 1 NO QAT DETECTED', [663].TIME.YEAR := 2016, [663].TIME.MONTH := 9, [663].TIME.DAY := 13, [663].TIME.HOUR := 9, [663].TIME.MINUTE := 8, [663].TIME.MICROSECOND := 699932, [663].EVENT := '2016/09/13   09:08:00   FAULT : Self Test 1 Charge (B-A) LOW', [664].TIME.YEAR := 2016, [664].TIME.MONTH := 9, [664].TIME.DAY := 13, [664].TIME.HOUR := 9, [664].TIME.MINUTE := 55, [664].TIME.SECOND := 54, [664].TIME.MICROSECOND := 899466, [664].EVENT := '2016/09/13   09:55:54   FAULT : QOW1 : Charge Outside Window Detected', [665].TIME.YEAR := 2016, [665].TIME.MONTH := 9, [665].TIME.DAY := 13, [665].TIME.HOUR := 9,
        [665].TIME.MINUTE := 55, [665].TIME.SECOND := 54, [665].TIME.MICROSECOND := 999842, [665].EVENT := '2016/09/13   09:55:54   FAULT : Self Test 2 Charge (B-A) HIGH', [666].TIME.YEAR := 2016, [666].TIME.MONTH := 9, [666].TIME.DAY := 13, [666].TIME.HOUR := 9, [666].TIME.MINUTE := 55, [666].TIME.SECOND := 55, [666].TIME.MICROSECOND := 499785, [666].EVENT := '2016/09/13   09:55:55   FAULT : Self Test 1 Charge (A-B) HIGH', [667].TIME.YEAR := 2016, [667].TIME.MONTH := 9, [667].TIME.DAY := 13, [667].TIME.HOUR := 9, [667].TIME.MINUTE := 55, [667].TIME.SECOND := 55, [667].TIME.MICROSECOND := 500347, [667].EVENT := '2016/09/13   09:55:55   FAULT : Self Test 1 B Baseline OUT OF RANGE', [668].TIME.YEAR := 2016, [668].TIME.MONTH := 9, [668].TIME.DAY := 13, [668].TIME.HOUR := 9, [668].TIME.MINUTE := 55, [668].TIME.SECOND := 55, [668].TIME.MICROSECOND := 999793, [668].EVENT := '2016/09/13   09:55:55   FAULT : Self Test 1 Charge (B-A) HIGH', [669].TIME.YEAR := 2016, [669].TIME.MONTH := 9, [669].TIME.DAY := 13, [669].TIME.HOUR := 9, [669].TIME.MINUTE := 55, [669].TIME.SECOND := 56, [669].TIME.MICROSECOND := 347, [669].EVENT := '2016/09/13   09:55:56   FAULT : Self Test 1 Charge (B-A) HIGH', [670].TIME.YEAR := 2016, [670].TIME.MONTH := 9, [670].TIME.DAY := 13, [670].TIME.HOUR := 9, [670].TIME.MINUTE := 55, [670].TIME.SECOND := 56, [670].TIME.MICROSECOND := 499836, [670].EVENT := '2016/09/13   09:55:56   FAULT : Self Test 2 Charge (A-B) HIGH', [671].TIME.YEAR := 2016, [671].TIME.MONTH := 9, [671].TIME.DAY := 13, [671].TIME.HOUR := 11, [671].TIME.MINUTE := 16, [671].TIME.SECOND := 54, [671].TIME.MICROSECOND := 199495, [671].EVENT := '2016/09/13   11:16:54   USER : RESET FAULT BUTTON PRESSED', [672].TIME.YEAR := 2016, [672].TIME.MONTH := 9, [672].TIME.DAY := 14, [672].TIME.HOUR := 9, [672].TIME.MINUTE := 42, [672].TIME.SECOND := 2, [672].TIME.MICROSECOND := 699531, [672].EVENT := '2016/09/14   09:42:02   USER : PPS RESET FAULT BUTTON PRESSED',
        [673].TIME.YEAR := 2016, [673].TIME.MONTH := 9, [673].TIME.DAY := 14, [673].TIME.HOUR := 9, [673].TIME.MINUTE := 42, [673].TIME.SECOND := 6, [673].TIME.MICROSECOND := 799506, [673].EVENT := '2016/09/14   09:42:06   USER : PPS RESET FAULT BUTTON PRESSED', [674].TIME.YEAR := 2016, [674].TIME.MONTH := 9, [674].TIME.DAY := 14, [674].TIME.HOUR := 9, [674].TIME.MINUTE := 42, [674].TIME.SECOND := 7, [674].TIME.MICROSECOND := 399506, [674].EVENT := '2016/09/14   09:42:07   USER : PPS RESET FAULT BUTTON PRESSED', [675].TIME.YEAR := 2016, [675].TIME.MONTH := 9, [675].TIME.DAY := 14, [675].TIME.HOUR := 9, [675].TIME.MINUTE := 42, [675].TIME.SECOND := 7, [675].TIME.MICROSECOND := 600025, [675].EVENT := '2016/09/14   09:42:07   USER : PPS RESET FAULT BUTTON PRESSED', [676].TIME.YEAR := 2016, [676].TIME.MONTH := 9, [676].TIME.DAY := 15, [676].TIME.HOUR := 10, [676].TIME.MINUTE := 18, [676].TIME.SECOND := 5, [676].TIME.MICROSECOND := 899467, [676].EVENT := '2016/09/15   10:18:05   USER : CERTIFICATION MODE ENABLED', [677].TIME.YEAR := 2016, [677].TIME.MONTH := 9, [677].TIME.DAY := 15, [677].TIME.HOUR := 10, [677].TIME.MINUTE := 18, [677].TIME.SECOND := 9, [677].TIME.MICROSECOND := 199998, [677].EVENT := '2016/09/15   10:18:09   USER : CERTIFICATION MODE DISABLED', [678].TIME.YEAR := 2016, [678].TIME.MONTH := 9, [678].TIME.DAY := 15, [678].TIME.HOUR := 10, [678].TIME.MINUTE := 36, [678].TIME.SECOND := 27, [678].TIME.MICROSECOND := 892487, [678].EVENT := '2016/09/15   10:36:27   USER : RESET FAULT BUTTON PRESSED', [679].TIME.YEAR := 2016, [679].TIME.MONTH := 9, [679].TIME.DAY := 20, [679].TIME.HOUR := 14, [679].TIME.MINUTE := 10, [679].TIME.SECOND := 53, [679].TIME.MICROSECOND := 692507, [679].EVENT := '2016/09/20   14:10:53   USER : PPS RESET FAULT BUTTON PRESSED', [680].TIME.YEAR := 2016, [680].TIME.MONTH := 9, [680].TIME.DAY := 20, [680].TIME.HOUR := 17,
        [680].TIME.MINUTE := 59, [680].TIME.SECOND := 54, [680].TIME.MICROSECOND := 92718, [680].EVENT := '2016/09/20   17:59:54   USER : PPS RESET FAULT BUTTON PRESSED', [681].TIME.YEAR := 2016, [681].TIME.MONTH := 9, [681].TIME.DAY := 21, [681].TIME.HOUR := 8, [681].TIME.MINUTE := 52, [681].TIME.SECOND := 34, [681].TIME.MICROSECOND := 92460, [681].EVENT := '2016/09/21   08:52:34   FAULT : QOW1 : Charge Outside Window Detected', [682].TIME.YEAR := 2016, [682].TIME.MONTH := 9, [682].TIME.DAY := 21, [682].TIME.HOUR := 8, [682].TIME.MINUTE := 52, [682].TIME.SECOND := 54, [682].TIME.MICROSECOND := 93017, [682].EVENT := '2016/09/21   08:52:54   USER : PPS RESET FAULT BUTTON PRESSED', [683].TIME.YEAR := 2016, [683].TIME.MONTH := 9, [683].TIME.DAY := 21, [683].TIME.HOUR := 10, [683].TIME.MINUTE := 30, [683].TIME.SECOND := 44, [683].TIME.MICROSECOND := 492504, [683].EVENT := '2016/09/21   10:30:44   USER : PPS RESET FAULT BUTTON PRESSED', [684].TIME.YEAR := 2016, [684].TIME.MONTH := 9, [684].TIME.DAY := 21, [684].TIME.HOUR := 10, [684].TIME.MINUTE := 32, [684].TIME.SECOND := 55, [684].TIME.MICROSECOND := 893023, [684].EVENT := '2016/09/21   10:32:55   USER : PPS RESET FAULT BUTTON PRESSED', [685].TIME.YEAR := 2016, [685].TIME.MONTH := 9, [685].TIME.DAY := 21, [685].TIME.HOUR := 10, [685].TIME.MINUTE := 33, [685].TIME.SECOND := 29, [685].TIME.MICROSECOND := 792499, [685].EVENT := '2016/09/21   10:33:29   USER : PPS RESET FAULT BUTTON PRESSED', [686].TIME.YEAR := 2016, [686].TIME.MONTH := 9, [686].TIME.DAY := 21, [686].TIME.HOUR := 11, [686].TIME.MINUTE := 5, [686].TIME.SECOND := 35, [686].TIME.MICROSECOND := 92507, [686].EVENT := '2016/09/21   11:05:35   USER : PPS RESET FAULT BUTTON PRESSED', [687].TIME.YEAR := 2016, [687].TIME.MONTH := 9, [687].TIME.DAY := 21, [687].TIME.HOUR := 11, [687].TIME.MINUTE := 5, [687].TIME.SECOND := 44, [687].TIME.MICROSECOND := 892938, [687].EVENT := '2016/09/21   11:05:44   USER : PPS RESET FAULT BUTTON PRESSED',
        [688].TIME.YEAR := 2016, [688].TIME.MONTH := 9, [688].TIME.DAY := 21, [688].TIME.HOUR := 11, [688].TIME.MINUTE := 5, [688].TIME.SECOND := 53, [688].TIME.MICROSECOND := 792501, [688].EVENT := '2016/09/21   11:05:53   USER : PPS RESET FAULT BUTTON PRESSED', [689].TIME.YEAR := 2016, [689].TIME.MONTH := 9, [689].TIME.DAY := 21, [689].TIME.HOUR := 11, [689].TIME.MINUTE := 19, [689].TIME.SECOND := 40, [689].TIME.MICROSECOND := 292459, [689].EVENT := '2016/09/21   11:19:40   FAULT : QOW1 : Charge Outside Window Detected', [690].TIME.YEAR := 2016, [690].TIME.MONTH := 9, [690].TIME.DAY := 21, [690].TIME.HOUR := 11, [690].TIME.MINUTE := 20, [690].TIME.SECOND := 1, [690].TIME.MICROSECOND := 92500, [690].EVENT := '2016/09/21   11:20:01   USER : PPS RESET FAULT BUTTON PRESSED', [691].TIME.YEAR := 2016, [691].TIME.MONTH := 9, [691].TIME.DAY := 21, [691].TIME.HOUR := 11, [691].TIME.MINUTE := 20, [691].TIME.SECOND := 2, [691].TIME.MICROSECOND := 792934, [691].EVENT := '2016/09/21   11:20:02   USER : PPS RESET FAULT BUTTON PRESSED', [692].TIME.YEAR := 2016, [692].TIME.MONTH := 9, [692].TIME.DAY := 21, [692].TIME.HOUR := 11, [692].TIME.MINUTE := 21, [692].TIME.SECOND := 40, [692].TIME.MICROSECOND := 192497, [692].EVENT := '2016/09/21   11:21:40   USER : PPS RESET FAULT BUTTON PRESSED', [693].TIME.YEAR := 2016, [693].TIME.MONTH := 9, [693].TIME.DAY := 21, [693].TIME.HOUR := 11, [693].TIME.MINUTE := 22, [693].TIME.SECOND := 25, [693].TIME.MICROSECOND := 992627, [693].EVENT := '2016/09/21   11:22:25   USER : PPS RESET FAULT BUTTON PRESSED', [694].TIME.YEAR := 2016, [694].TIME.MONTH := 9, [694].TIME.DAY := 21, [694].TIME.HOUR := 11, [694].TIME.MINUTE := 22, [694].TIME.SECOND := 27, [694].TIME.MICROSECOND := 492933, [694].EVENT := '2016/09/21   11:22:27   USER : PPS RESET FAULT BUTTON PRESSED', [695].TIME.YEAR := 2016, [695].TIME.MONTH := 9, [695].TIME.DAY := 21, [695].TIME.HOUR := 11,
        [695].TIME.MINUTE := 22, [695].TIME.SECOND := 38, [695].TIME.MICROSECOND := 192934, [695].EVENT := '2016/09/21   11:22:38   USER : PPS RESET FAULT BUTTON PRESSED', [696].TIME.YEAR := 2016, [696].TIME.MONTH := 9, [696].TIME.DAY := 21, [696].TIME.HOUR := 11, [696].TIME.MINUTE := 35, [696].TIME.SECOND := 37, [696].TIME.MICROSECOND := 692644, [696].EVENT := '2016/09/21   11:35:37   USER : BYPASS KEY SET TO ENABLE', [697].TIME.YEAR := 2016, [697].TIME.MONTH := 9, [697].TIME.DAY := 21, [697].TIME.HOUR := 11, [697].TIME.MINUTE := 36, [697].TIME.SECOND := 53, [697].TIME.MICROSECOND := 192514, [697].EVENT := '2016/09/21   11:36:53   USER : BYPASS KEY SET TO DISABLE', [698].TIME.YEAR := 2016, [698].TIME.MONTH := 9, [698].TIME.DAY := 21, [698].TIME.HOUR := 11, [698].TIME.MINUTE := 36, [698].TIME.SECOND := 55, [698].TIME.MICROSECOND := 592937, [698].EVENT := '2016/09/21   11:36:55   USER : BYPASS KEY SET TO ENABLE', [699].TIME.YEAR := 2016, [699].TIME.MONTH := 9, [699].TIME.DAY := 21, [699].TIME.HOUR := 11, [699].TIME.MINUTE := 36, [699].TIME.SECOND := 56, [699].TIME.MICROSECOND := 892510, [699].EVENT := '2016/09/21   11:36:56   USER : BYPASS KEY SET TO DISABLE', [700].TIME.YEAR := 2016, [700].TIME.MONTH := 9, [700].TIME.DAY := 21, [700].TIME.HOUR := 11, [700].TIME.MINUTE := 36, [700].TIME.SECOND := 57, [700].TIME.MICROSECOND := 592939, [700].EVENT := '2016/09/21   11:36:57   USER : BYPASS KEY SET TO ENABLE', [701].TIME.YEAR := 2016, [701].TIME.MONTH := 9, [701].TIME.DAY := 21, [701].TIME.HOUR := 11, [701].TIME.MINUTE := 36, [701].TIME.SECOND := 58, [701].TIME.MICROSECOND := 192506, [701].EVENT := '2016/09/21   11:36:58   USER : BYPASS KEY SET TO DISABLE', [702].TIME.YEAR := 2016, [702].TIME.MONTH := 9, [702].TIME.DAY := 21, [702].TIME.HOUR := 11, [702].TIME.MINUTE := 36, [702].TIME.SECOND := 58, [702].TIME.MICROSECOND := 692507, [702].EVENT := '2016/09/21   11:36:58   USER : BYPASS KEY SET TO ENABLE',
        [703].TIME.YEAR := 2016, [703].TIME.MONTH := 9, [703].TIME.DAY := 21, [703].TIME.HOUR := 11, [703].TIME.MINUTE := 36, [703].TIME.SECOND := 59, [703].TIME.MICROSECOND := 492513, [703].EVENT := '2016/09/21   11:36:59   USER : BYPASS KEY SET TO DISABLE', [704].TIME.YEAR := 2016, [704].TIME.MONTH := 9, [704].TIME.DAY := 21, [704].TIME.HOUR := 11, [704].TIME.MINUTE := 36, [704].TIME.SECOND := 59, [704].TIME.MICROSECOND := 992509, [704].EVENT := '2016/09/21   11:36:59   USER : BYPASS KEY SET TO ENABLE', [705].TIME.YEAR := 2016, [705].TIME.MONTH := 9, [705].TIME.DAY := 21, [705].TIME.HOUR := 11, [705].TIME.MINUTE := 37, [705].TIME.SECOND := 1, [705].TIME.MICROSECOND := 292511, [705].EVENT := '2016/09/21   11:37:01   USER : BYPASS KEY SET TO DISABLE', [706].TIME.YEAR := 2016, [706].TIME.MONTH := 9, [706].TIME.DAY := 21, [706].TIME.HOUR := 11, [706].TIME.MINUTE := 37, [706].TIME.SECOND := 4, [706].TIME.MICROSECOND := 92518, [706].EVENT := '2016/09/21   11:37:04   USER : BYPASS KEY SET TO ENABLE', [707].TIME.YEAR := 2016, [707].TIME.MONTH := 9, [707].TIME.DAY := 21, [707].TIME.HOUR := 11, [707].TIME.MINUTE := 43, [707].TIME.SECOND := 15, [707].TIME.MICROSECOND := 192503, [707].EVENT := '2016/09/21   11:43:15   USER : PPS RESET FAULT BUTTON PRESSED', [708].TIME.YEAR := 2016, [708].TIME.MONTH := 9, [708].TIME.DAY := 21, [708].TIME.HOUR := 11, [708].TIME.MINUTE := 44, [708].TIME.SECOND := 2, [708].TIME.MICROSECOND := 592529, [708].EVENT := '2016/09/21   11:44:02   USER : BYPASS KEY SET TO DISABLE', [709].TIME.YEAR := 2016, [709].TIME.MONTH := 9, [709].TIME.DAY := 21, [709].TIME.HOUR := 11, [709].TIME.MINUTE := 51, [709].TIME.SECOND := 50, [709].TIME.MICROSECOND := 392485, [709].EVENT := '2016/09/21   11:51:50   FAULT : QOW1 : Charge Outside Window Detected', [710].TIME.YEAR := 2016, [710].TIME.MONTH := 9, [710].TIME.DAY := 21, [710].TIME.HOUR := 11,
        [710].TIME.MINUTE := 53, [710].TIME.SECOND := 14, [710].TIME.MICROSECOND := 193076, [710].EVENT := '2016/09/21   11:53:14   USER : PPS RESET FAULT BUTTON PRESSED', [711].TIME.YEAR := 2016, [711].TIME.MONTH := 9, [711].TIME.DAY := 21, [711].TIME.HOUR := 11, [711].TIME.MINUTE := 53, [711].TIME.SECOND := 56, [711].TIME.MICROSECOND := 92510, [711].EVENT := '2016/09/21   11:53:56   USER : PPS RESET FAULT BUTTON PRESSED', [712].TIME.YEAR := 2016, [712].TIME.MONTH := 9, [712].TIME.DAY := 21, [712].TIME.HOUR := 13, [712].TIME.MINUTE := 10, [712].TIME.SECOND := 40, [712].TIME.MICROSECOND := 292456, [712].EVENT := '2016/09/21   13:10:40   FAULT : QOW1 : Charge Outside Window Detected', [713].TIME.YEAR := 2016, [713].TIME.MONTH := 9, [713].TIME.DAY := 21, [713].TIME.HOUR := 13, [713].TIME.MINUTE := 15, [713].TIME.SECOND := 57, [713].TIME.MICROSECOND := 592486, [713].EVENT := '2016/09/21   13:15:57   USER : RESET FAULT BUTTON PRESSED', [714].TIME.YEAR := 2016, [714].TIME.MONTH := 9, [714].TIME.DAY := 21, [714].TIME.HOUR := 13, [714].TIME.MINUTE := 17, [714].TIME.SECOND := 53, [714].TIME.MICROSECOND := 592455, [714].EVENT := '2016/09/21   13:17:53   FAULT : QOW1 : Charge Outside Window Detected', [715].TIME.YEAR := 2016, [715].TIME.MONTH := 9, [715].TIME.DAY := 21, [715].TIME.HOUR := 13, [715].TIME.MINUTE := 17, [715].TIME.SECOND := 54, [715].TIME.MICROSECOND := 492509, [715].EVENT := '2016/09/21   13:17:54   USER : PPS RESET FAULT BUTTON PRESSED', [716].TIME.YEAR := 2016, [716].TIME.MONTH := 9, [716].TIME.DAY := 21, [716].TIME.HOUR := 13, [716].TIME.MINUTE := 37, [716].TIME.SECOND := 59, [716].TIME.MICROSECOND := 92507, [716].EVENT := '2016/09/21   13:37:59   USER : PPS RESET FAULT BUTTON PRESSED', [717].TIME.YEAR := 2016, [717].TIME.MONTH := 9, [717].TIME.DAY := 21, [717].TIME.HOUR := 13, [717].TIME.MINUTE := 38, [717].TIME.SECOND := 52, [717].TIME.MICROSECOND := 693101, [717].EVENT := '2016/09/21   13:38:52   FAULT : QOW1 : Charge Outside Window Detected',
        [718].TIME.YEAR := 2016, [718].TIME.MONTH := 9, [718].TIME.DAY := 21, [718].TIME.HOUR := 13, [718].TIME.MINUTE := 38, [718].TIME.SECOND := 53, [718].TIME.MICROSECOND := 592500, [718].EVENT := '2016/09/21   13:38:53   USER : PPS RESET FAULT BUTTON PRESSED', [719].TIME.YEAR := 2016, [719].TIME.MONTH := 9, [719].TIME.DAY := 21, [719].TIME.HOUR := 13, [719].TIME.MINUTE := 39, [719].TIME.SECOND := 31, [719].TIME.MICROSECOND := 92626, [719].EVENT := '2016/09/21   13:39:31   USER : PPS RESET FAULT BUTTON PRESSED', [720].TIME.YEAR := 2016, [720].TIME.MONTH := 9, [720].TIME.DAY := 21, [720].TIME.HOUR := 13, [720].TIME.MINUTE := 52, [720].TIME.SECOND := 50, [720].TIME.MICROSECOND := 392500, [720].EVENT := '2016/09/21   13:52:50   USER : PPS RESET FAULT BUTTON PRESSED', [721].TIME.YEAR := 2016, [721].TIME.MONTH := 9, [721].TIME.DAY := 21, [721].TIME.HOUR := 13, [721].TIME.MINUTE := 52, [721].TIME.SECOND := 54, [721].TIME.MICROSECOND := 293032, [721].EVENT := '2016/09/21   13:52:54   USER : PPS RESET FAULT BUTTON PRESSED', [722].TIME.YEAR := 2016, [722].TIME.MONTH := 9, [722].TIME.DAY := 21, [722].TIME.HOUR := 16, [722].TIME.MINUTE := 41, [722].TIME.SECOND := 45, [722].TIME.MICROSECOND := 992458, [722].EVENT := '2016/09/21   16:41:45   FAULT : QOW1 : Charge Outside Window Detected', [723].TIME.YEAR := 2016, [723].TIME.MONTH := 9, [723].TIME.DAY := 21, [723].TIME.HOUR := 16, [723].TIME.MINUTE := 41, [723].TIME.SECOND := 46, [723].TIME.MICROSECOND := 292505, [723].EVENT := '2016/09/21   16:41:46   USER : PPS RESET FAULT BUTTON PRESSED', [724].TIME.YEAR := 2016, [724].TIME.MONTH := 9, [724].TIME.DAY := 21, [724].TIME.HOUR := 17, [724].TIME.MINUTE := 22, [724].TIME.SECOND := 5, [724].TIME.MICROSECOND := 692509, [724].EVENT := '2016/09/21   17:22:05   USER : PPS RESET FAULT BUTTON PRESSED', [725].TIME.YEAR := 2016, [725].TIME.MONTH := 9, [725].TIME.DAY := 21, [725].TIME.HOUR := 17,
        [725].TIME.MINUTE := 22, [725].TIME.SECOND := 20, [725].TIME.MICROSECOND := 692504, [725].EVENT := '2016/09/21   17:22:20   USER : PPS RESET FAULT BUTTON PRESSED', [726].TIME.YEAR := 2016, [726].TIME.MONTH := 9, [726].TIME.DAY := 21, [726].TIME.HOUR := 17, [726].TIME.MINUTE := 23, [726].TIME.SECOND := 7, [726].TIME.MICROSECOND := 92508, [726].EVENT := '2016/09/21   17:23:07   USER : PPS RESET FAULT BUTTON PRESSED', [727].TIME.YEAR := 2016, [727].TIME.MONTH := 9, [727].TIME.DAY := 22, [727].TIME.HOUR := 10, [727].TIME.MINUTE := 41, [727].TIME.SECOND := 28, [727].TIME.MICROSECOND := 392502, [727].EVENT := '2016/09/22   10:41:28   USER : PPS RESET FAULT BUTTON PRESSED', [728].TIME.YEAR := 2016, [728].TIME.MONTH := 9, [728].TIME.DAY := 22, [728].TIME.HOUR := 10, [728].TIME.MINUTE := 57, [728].TIME.SECOND := 32, [728].TIME.MICROSECOND := 892458, [728].EVENT := '2016/09/22   10:57:32   FAULT : QOW1 : Charge Outside Window Detected', [729].TIME.YEAR := 2016, [729].TIME.MONTH := 9, [729].TIME.DAY := 22, [729].TIME.HOUR := 11, [729].TIME.SECOND := 46, [729].TIME.MICROSECOND := 492502, [729].EVENT := '2016/09/22   11:00:46   USER : PPS RESET FAULT BUTTON PRESSED', [730].TIME.YEAR := 2016, [730].TIME.MONTH := 9, [730].TIME.DAY := 22, [730].TIME.HOUR := 11, [730].TIME.MINUTE := 4, [730].TIME.SECOND := 43, [730].TIME.MICROSECOND := 392509, [730].EVENT := '2016/09/22   11:04:43   USER : BYPASS KEY SET TO ENABLE', [731].TIME.YEAR := 2016, [731].TIME.MONTH := 9, [731].TIME.DAY := 22, [731].TIME.HOUR := 11, [731].TIME.MINUTE := 4, [731].TIME.SECOND := 51, [731].TIME.MICROSECOND := 492555, [731].EVENT := '2016/09/22   11:04:51   USER : PPS RESET FAULT BUTTON PRESSED', [732].TIME.YEAR := 2016, [732].TIME.MONTH := 9, [732].TIME.DAY := 22, [732].TIME.HOUR := 11, [732].TIME.MINUTE := 4, [732].TIME.SECOND := 52, [732].TIME.MICROSECOND := 893024, [732].EVENT := '2016/09/22   11:04:52   USER : PPS RESET FAULT BUTTON PRESSED', [733].TIME.YEAR := 2016,
        [733].TIME.MONTH := 9, [733].TIME.DAY := 22, [733].TIME.HOUR := 11, [733].TIME.MINUTE := 4, [733].TIME.SECOND := 53, [733].TIME.MICROSECOND := 492515, [733].EVENT := '2016/09/22   11:04:53   USER : PPS RESET FAULT BUTTON PRESSED', [734].TIME.YEAR := 2016, [734].TIME.MONTH := 9, [734].TIME.DAY := 22, [734].TIME.HOUR := 11, [734].TIME.MINUTE := 4, [734].TIME.SECOND := 54, [734].TIME.MICROSECOND := 192500, [734].EVENT := '2016/09/22   11:04:54   USER : PPS RESET FAULT BUTTON PRESSED', [735].TIME.YEAR := 2016, [735].TIME.MONTH := 9, [735].TIME.DAY := 22, [735].TIME.HOUR := 11, [735].TIME.MINUTE := 8, [735].TIME.SECOND := 35, [735].TIME.MICROSECOND := 792505, [735].EVENT := '2016/09/22   11:08:35   USER : PPS RESET FAULT BUTTON PRESSED', [736].TIME.YEAR := 2016, [736].TIME.MONTH := 9, [736].TIME.DAY := 22, [736].TIME.HOUR := 11, [736].TIME.MINUTE := 13, [736].TIME.SECOND := 15, [736].TIME.MICROSECOND := 892457, [736].EVENT := '2016/09/22   11:13:15   FAULT : QOW1 : Charge Outside Window Detected', [737].TIME.YEAR := 2016, [737].TIME.MONTH := 9, [737].TIME.DAY := 22, [737].TIME.HOUR := 11, [737].TIME.MINUTE := 15, [737].TIME.SECOND := 48, [737].TIME.MICROSECOND := 392507, [737].EVENT := '2016/09/22   11:15:48   USER : PPS RESET FAULT BUTTON PRESSED', [738].TIME.YEAR := 2016, [738].TIME.MONTH := 9, [738].TIME.DAY := 22, [738].TIME.HOUR := 11, [738].TIME.MINUTE := 20, [738].TIME.SECOND := 54, [738].TIME.MICROSECOND := 492507, [738].EVENT := '2016/09/22   11:20:54   USER : PPS RESET FAULT BUTTON PRESSED', [739].TIME.YEAR := 2016, [739].TIME.MONTH := 9, [739].TIME.DAY := 22, [739].TIME.HOUR := 13, [739].TIME.MINUTE := 15, [739].TIME.SECOND := 59, [739].TIME.MICROSECOND := 992455, [739].EVENT := '2016/09/22   13:15:59   FAULT : QOW1 : Charge Outside Window Detected', [740].TIME.YEAR := 2016, [740].TIME.MONTH := 9, [740].TIME.DAY := 22, [740].TIME.HOUR := 13, [740].TIME.MINUTE := 16,
        [740].TIME.MICROSECOND := 292503, [740].EVENT := '2016/09/22   13:16:00   USER : PPS RESET FAULT BUTTON PRESSED', [741].TIME.YEAR := 2016, [741].TIME.MONTH := 9, [741].TIME.DAY := 22, [741].TIME.HOUR := 13, [741].TIME.MINUTE := 16, [741].TIME.SECOND := 1, [741].TIME.MICROSECOND := 392543, [741].EVENT := '2016/09/22   13:16:01   USER : PPS RESET FAULT BUTTON PRESSED', [742].TIME.YEAR := 2016, [742].TIME.MONTH := 9, [742].TIME.DAY := 22, [742].TIME.HOUR := 13, [742].TIME.MINUTE := 16, [742].TIME.SECOND := 2, [742].TIME.MICROSECOND := 793023, [742].EVENT := '2016/09/22   13:16:02   USER : PPS RESET FAULT BUTTON PRESSED', [743].TIME.YEAR := 2016, [743].TIME.MONTH := 9, [743].TIME.DAY := 22, [743].TIME.HOUR := 13, [743].TIME.MINUTE := 26, [743].TIME.SECOND := 17, [743].TIME.MICROSECOND := 892506, [743].EVENT := '2016/09/22   13:26:17   USER : PPS RESET FAULT BUTTON PRESSED', [744].TIME.YEAR := 2016, [744].TIME.MONTH := 9, [744].TIME.DAY := 22, [744].TIME.HOUR := 13, [744].TIME.MINUTE := 26, [744].TIME.SECOND := 22, [744].TIME.MICROSECOND := 292978, [744].EVENT := '2016/09/22   13:26:22   FAULT : QOW1 : Charge Outside Window Detected', [745].TIME.YEAR := 2016, [745].TIME.MONTH := 9, [745].TIME.DAY := 22, [745].TIME.HOUR := 13, [745].TIME.MINUTE := 26, [745].TIME.SECOND := 24, [745].TIME.MICROSECOND := 192517, [745].EVENT := '2016/09/22   13:26:24   USER : PPS RESET FAULT BUTTON PRESSED', [746].TIME.YEAR := 2016, [746].TIME.MONTH := 9, [746].TIME.DAY := 22, [746].TIME.HOUR := 13, [746].TIME.MINUTE := 32, [746].TIME.SECOND := 35, [746].TIME.MICROSECOND := 792450, [746].EVENT := '2016/09/22   13:32:35   FAULT : QOW1 : Charge Outside Window Detected', [747].TIME.YEAR := 2016, [747].TIME.MONTH := 9, [747].TIME.DAY := 22, [747].TIME.HOUR := 13, [747].TIME.MINUTE := 32, [747].TIME.SECOND := 35, [747].TIME.MICROSECOND := 992507, [747].EVENT := '2016/09/22   13:32:35   USER : PPS RESET FAULT BUTTON PRESSED', [748].TIME.YEAR := 2016, [748].TIME.MONTH := 9,
        [748].TIME.DAY := 22, [748].TIME.HOUR := 13, [748].TIME.MINUTE := 35, [748].TIME.SECOND := 28, [748].TIME.MICROSECOND := 592515, [748].EVENT := '2016/09/22   13:35:28   USER : PPS RESET FAULT BUTTON PRESSED', [749].TIME.YEAR := 2016, [749].TIME.MONTH := 9, [749].TIME.DAY := 22, [749].TIME.HOUR := 13, [749].TIME.MINUTE := 35, [749].TIME.SECOND := 47, [749].TIME.MICROSECOND := 392468, [749].EVENT := '2016/09/22   13:35:47   FAULT : QOW1 : Charge Outside Window Detected', [750].TIME.YEAR := 2016, [750].TIME.MONTH := 9, [750].TIME.DAY := 22, [750].TIME.HOUR := 13, [750].TIME.MINUTE := 40, [750].TIME.SECOND := 30, [750].TIME.MICROSECOND := 692509, [750].EVENT := '2016/09/22   13:40:30   USER : PPS RESET FAULT BUTTON PRESSED', [751].TIME.YEAR := 2016, [751].TIME.MONTH := 9, [751].TIME.DAY := 22, [751].TIME.HOUR := 13, [751].TIME.MINUTE := 41, [751].TIME.SECOND := 32, [751].TIME.MICROSECOND := 592497, [751].EVENT := '2016/09/22   13:41:32   USER : PPS RESET FAULT BUTTON PRESSED', [752].TIME.YEAR := 2016, [752].TIME.MONTH := 9, [752].TIME.DAY := 22, [752].TIME.HOUR := 13, [752].TIME.MINUTE := 46, [752].TIME.SECOND := 20, [752].TIME.MICROSECOND := 492993, [752].EVENT := '2016/09/22   13:46:20   FAULT : QOW1 : Charge Outside Window Detected', [753].TIME.YEAR := 2016, [753].TIME.MONTH := 9, [753].TIME.DAY := 22, [753].TIME.HOUR := 13, [753].TIME.MINUTE := 46, [753].TIME.SECOND := 20, [753].TIME.MICROSECOND := 792646, [753].EVENT := '2016/09/22   13:46:20   USER : PPS RESET FAULT BUTTON PRESSED', [754].TIME.YEAR := 2016, [754].TIME.MONTH := 9, [754].TIME.DAY := 22, [754].TIME.HOUR := 13, [754].TIME.MINUTE := 47, [754].TIME.SECOND := 57, [754].TIME.MICROSECOND := 192499, [754].EVENT := '2016/09/22   13:47:57   USER : PPS RESET FAULT BUTTON PRESSED', [755].TIME.YEAR := 2016, [755].TIME.MONTH := 9, [755].TIME.DAY := 22, [755].TIME.HOUR := 13, [755].TIME.MINUTE := 48, [755].TIME.SECOND := 8,
